    CONST robtarget T669:=[[77.479995,87.050626,11.799995],[0.000000,0.000000,1.000000,0.000000],[0,0,-1,0],[9E+09,9E+09,9E+09,9E+09,9E+09,9E+09]];
    CONST robtarget T670:=[[77.479995,72.949381,11.799995],[0.000000,0.000000,1.000000,0.000000],[0,0,-1,0],[9E+09,9E+09,9E+09,9E+09,9E+09,9E+09]];
    CONST robtarget T671:=[[77.479995,52.050624,11.799995],[0.000000,0.000000,1.000000,0.000000],[0,0,-1,0],[9E+09,9E+09,9E+09,9E+09,9E+09,9E+09]];
    CONST robtarget T672:=[[77.479995,37.949379,11.799995],[0.000000,0.000000,1.000000,0.000000],[0,0,-1,0],[9E+09,9E+09,9E+09,9E+09,9E+09,9E+09]];
    CONST robtarget T673:=[[77.479995,30.069007,11.799995],[0.000000,0.000000,1.000000,0.000000],[0,0,-1,0],[9E+09,9E+09,9E+09,9E+09,9E+09,9E+09]];
    CONST robtarget T674:=[[78.739999,30.028279,11.799995],[0.000000,0.000000,1.000000,0.000000],[0,0,-1,0],[9E+09,9E+09,9E+09,9E+09,9E+09,9E+09]];
    CONST robtarget T675:=[[78.739999,37.608991,11.799995],[0.000000,0.000000,1.000000,0.000000],[0,0,-1,0],[9E+09,9E+09,9E+09,9E+09,9E+09,9E+09]];
    CONST robtarget T676:=[[78.739999,52.391011,11.799995],[0.000000,0.000000,1.000000,0.000000],[0,0,-1,0],[9E+09,9E+09,9E+09,9E+09,9E+09,9E+09]];
    CONST robtarget T677:=[[78.739999,72.608994,11.799995],[0.000000,0.000000,1.000000,0.000000],[0,0,-1,0],[9E+09,9E+09,9E+09,9E+09,9E+09,9E+09]];
    CONST robtarget T678:=[[78.739999,87.391014,11.799995],[0.000000,0.000000,1.000000,0.000000],[0,0,-1,0],[9E+09,9E+09,9E+09,9E+09,9E+09,9E+09]];
    CONST robtarget T679:=[[78.739999,107.608996,11.799995],[0.000000,0.000000,1.000000,0.000000],[0,0,-1,0],[9E+09,9E+09,9E+09,9E+09,9E+09,9E+09]];
    CONST robtarget T680:=[[78.739999,122.391017,11.799995],[0.000000,0.000000,1.000000,0.000000],[0,0,-1,0],[9E+09,9E+09,9E+09,9E+09,9E+09,9E+09]];
    CONST robtarget T681:=[[78.739999,129.971729,11.799995],[0.000000,0.000000,1.000000,0.000000],[0,0,-1,0],[9E+09,9E+09,9E+09,9E+09,9E+09,9E+09]];
    CONST robtarget T682:=[[80.000004,130.000008,11.799995],[0.000000,0.000000,1.000000,0.000000],[0,0,-1,0],[9E+09,9E+09,9E+09,9E+09,9E+09,9E+09]];
    CONST robtarget T683:=[[80.000004,122.487319,11.799995],[0.000000,0.000000,1.000000,0.000000],[0,0,-1,0],[9E+09,9E+09,9E+09,9E+09,9E+09,9E+09]];
    CONST robtarget T684:=[[80.000004,107.512696,11.799995],[0.000000,0.000000,1.000000,0.000000],[0,0,-1,0],[9E+09,9E+09,9E+09,9E+09,9E+09,9E+09]];
    CONST robtarget T685:=[[80.000004,87.487316,11.799995],[0.000000,0.000000,1.000000,0.000000],[0,0,-1,0],[9E+09,9E+09,9E+09,9E+09,9E+09,9E+09]];
    CONST robtarget T686:=[[80.000004,72.512692,11.799995],[0.000000,0.000000,1.000000,0.000000],[0,0,-1,0],[9E+09,9E+09,9E+09,9E+09,9E+09,9E+09]];
    CONST robtarget T687:=[[80.000004,52.487312,11.799995],[0.000000,0.000000,1.000000,0.000000],[0,0,-1,0],[9E+09,9E+09,9E+09,9E+09,9E+09,9E+09]];
    CONST robtarget T688:=[[80.000004,37.512688,11.799995],[0.000000,0.000000,1.000000,0.000000],[0,0,-1,0],[9E+09,9E+09,9E+09,9E+09,9E+09,9E+09]];
    CONST robtarget T689:=[[80.000004,30.000000,11.799995],[0.000000,0.000000,1.000000,0.000000],[0,0,-1,0],[9E+09,9E+09,9E+09,9E+09,9E+09,9E+09]];
    CONST robtarget T690:=[[81.260008,30.028279,11.799995],[0.000000,0.000000,1.000000,0.000000],[0,0,-1,0],[9E+09,9E+09,9E+09,9E+09,9E+09,9E+09]];
    CONST robtarget T691:=[[81.260008,37.608991,11.799995],[0.000000,0.000000,1.000000,0.000000],[0,0,-1,0],[9E+09,9E+09,9E+09,9E+09,9E+09,9E+09]];
    CONST robtarget T692:=[[81.260008,52.391011,11.799995],[0.000000,0.000000,1.000000,0.000000],[0,0,-1,0],[9E+09,9E+09,9E+09,9E+09,9E+09,9E+09]];
    CONST robtarget T693:=[[81.260008,72.608994,11.799995],[0.000000,0.000000,1.000000,0.000000],[0,0,-1,0],[9E+09,9E+09,9E+09,9E+09,9E+09,9E+09]];
    CONST robtarget T694:=[[81.260008,87.391014,11.799995],[0.000000,0.000000,1.000000,0.000000],[0,0,-1,0],[9E+09,9E+09,9E+09,9E+09,9E+09,9E+09]];
    CONST robtarget T695:=[[81.260008,107.608996,11.799995],[0.000000,0.000000,1.000000,0.000000],[0,0,-1,0],[9E+09,9E+09,9E+09,9E+09,9E+09,9E+09]];
    CONST robtarget T696:=[[81.260008,122.391017,11.799995],[0.000000,0.000000,1.000000,0.000000],[0,0,-1,0],[9E+09,9E+09,9E+09,9E+09,9E+09,9E+09]];
    CONST robtarget T697:=[[81.260008,129.971729,11.799995],[0.000000,0.000000,1.000000,0.000000],[0,0,-1,0],[9E+09,9E+09,9E+09,9E+09,9E+09,9E+09]];
    CONST robtarget T698:=[[82.520013,129.931001,11.799995],[0.000000,0.000000,1.000000,0.000000],[0,0,-1,0],[9E+09,9E+09,9E+09,9E+09,9E+09,9E+09]];
    CONST robtarget T699:=[[82.520013,122.050628,11.799995],[0.000000,0.000000,1.000000,0.000000],[0,0,-1,0],[9E+09,9E+09,9E+09,9E+09,9E+09,9E+09]];
    CONST robtarget T700:=[[82.520013,107.949384,11.799995],[0.000000,0.000000,1.000000,0.000000],[0,0,-1,0],[9E+09,9E+09,9E+09,9E+09,9E+09,9E+09]];
    CONST robtarget T701:=[[82.520013,87.050626,11.799995],[0.000000,0.000000,1.000000,0.000000],[0,0,-1,0],[9E+09,9E+09,9E+09,9E+09,9E+09,9E+09]];
    CONST robtarget T702:=[[82.520013,72.949381,11.799995],[0.000000,0.000000,1.000000,0.000000],[0,0,-1,0],[9E+09,9E+09,9E+09,9E+09,9E+09,9E+09]];
    CONST robtarget T703:=[[82.520013,52.050624,11.799995],[0.000000,0.000000,1.000000,0.000000],[0,0,-1,0],[9E+09,9E+09,9E+09,9E+09,9E+09,9E+09]];
    CONST robtarget T704:=[[82.520013,37.949379,11.799995],[0.000000,0.000000,1.000000,0.000000],[0,0,-1,0],[9E+09,9E+09,9E+09,9E+09,9E+09,9E+09]];
    CONST robtarget T705:=[[82.520013,30.069007,11.799995],[0.000000,0.000000,1.000000,0.000000],[0,0,-1,0],[9E+09,9E+09,9E+09,9E+09,9E+09,9E+09]];
    CONST robtarget T706:=[[83.780017,30.153959,11.799995],[0.000000,0.000000,1.000000,0.000000],[0,0,-1,0],[9E+09,9E+09,9E+09,9E+09,9E+09,9E+09]];
    CONST robtarget T707:=[[83.780017,38.524551,11.799995],[0.000000,0.000000,1.000000,0.000000],[0,0,-1,0],[9E+09,9E+09,9E+09,9E+09,9E+09,9E+09]];
    CONST robtarget T708:=[[83.780017,51.475451,11.799995],[0.000000,0.000000,1.000000,0.000000],[0,0,-1,0],[9E+09,9E+09,9E+09,9E+09,9E+09,9E+09]];
    CONST robtarget T709:=[[83.780017,73.524553,11.799995],[0.000000,0.000000,1.000000,0.000000],[0,0,-1,0],[9E+09,9E+09,9E+09,9E+09,9E+09,9E+09]];
    CONST robtarget T710:=[[83.780017,86.475455,11.799995],[0.000000,0.000000,1.000000,0.000000],[0,0,-1,0],[9E+09,9E+09,9E+09,9E+09,9E+09,9E+09]];
    CONST robtarget T711:=[[83.780017,108.524556,11.799995],[0.000000,0.000000,1.000000,0.000000],[0,0,-1,0],[9E+09,9E+09,9E+09,9E+09,9E+09,9E+09]];
    CONST robtarget T712:=[[83.780017,121.475457,11.799995],[0.000000,0.000000,1.000000,0.000000],[0,0,-1,0],[9E+09,9E+09,9E+09,9E+09,9E+09,9E+09]];
    CONST robtarget T713:=[[83.780017,129.846049,11.799995],[0.000000,0.000000,1.000000,0.000000],[0,0,-1,0],[9E+09,9E+09,9E+09,9E+09,9E+09,9E+09]];
    CONST robtarget T714:=[[85.040022,129.735844,11.799995],[0.000000,0.000000,1.000000,0.000000],[0,0,-1,0],[9E+09,9E+09,9E+09,9E+09,9E+09,9E+09]];
    CONST robtarget T715:=[[85.040022,120.544921,11.799995],[0.000000,0.000000,1.000000,0.000000],[0,0,-1,0],[9E+09,9E+09,9E+09,9E+09,9E+09,9E+09]];
    CONST robtarget T716:=[[85.040022,109.455091,11.799995],[0.000000,0.000000,1.000000,0.000000],[0,0,-1,0],[9E+09,9E+09,9E+09,9E+09,9E+09,9E+09]];
    CONST robtarget T717:=[[85.040022,85.544918,11.799995],[0.000000,0.000000,1.000000,0.000000],[0,0,-1,0],[9E+09,9E+09,9E+09,9E+09,9E+09,9E+09]];
    CONST robtarget T718:=[[85.040022,74.455090,11.799995],[0.000000,0.000000,1.000000,0.000000],[0,0,-1,0],[9E+09,9E+09,9E+09,9E+09,9E+09,9E+09]];
    CONST robtarget T719:=[[85.040022,50.544916,11.799995],[0.000000,0.000000,1.000000,0.000000],[0,0,-1,0],[9E+09,9E+09,9E+09,9E+09,9E+09,9E+09]];
    CONST robtarget T720:=[[85.040022,39.455086,11.799995],[0.000000,0.000000,1.000000,0.000000],[0,0,-1,0],[9E+09,9E+09,9E+09,9E+09,9E+09,9E+09]];
    CONST robtarget T721:=[[85.040022,30.264163,11.799995],[0.000000,0.000000,1.000000,0.000000],[0,0,-1,0],[9E+09,9E+09,9E+09,9E+09,9E+09,9E+09]];
    CONST robtarget T722:=[[86.300026,30.406130,11.799995],[0.000000,0.000000,1.000000,0.000000],[0,0,-1,0],[9E+09,9E+09,9E+09,9E+09,9E+09,9E+09]];
    CONST robtarget T723:=[[86.300026,40.937335,11.799995],[0.000000,0.000000,1.000000,0.000000],[0,0,-1,0],[9E+09,9E+09,9E+09,9E+09,9E+09,9E+09]];
    CONST robtarget T724:=[[86.300026,49.062665,11.799995],[0.000000,0.000000,1.000000,0.000000],[0,0,-1,0],[9E+09,9E+09,9E+09,9E+09,9E+09,9E+09]];
    CONST robtarget T725:=[[86.300026,75.937339,11.799995],[0.000000,0.000000,1.000000,0.000000],[0,0,-1,0],[9E+09,9E+09,9E+09,9E+09,9E+09,9E+09]];
    CONST robtarget T726:=[[86.300026,84.062668,11.799995],[0.000000,0.000000,1.000000,0.000000],[0,0,-1,0],[9E+09,9E+09,9E+09,9E+09,9E+09,9E+09]];
    CONST robtarget T727:=[[86.300026,110.937342,11.799995],[0.000000,0.000000,1.000000,0.000000],[0,0,-1,0],[9E+09,9E+09,9E+09,9E+09,9E+09,9E+09]];
    CONST robtarget T728:=[[86.300026,119.062672,11.799995],[0.000000,0.000000,1.000000,0.000000],[0,0,-1,0],[9E+09,9E+09,9E+09,9E+09,9E+09,9E+09]];
    CONST robtarget T729:=[[86.300026,129.593877,11.799995],[0.000000,0.000000,1.000000,0.000000],[0,0,-1,0],[9E+09,9E+09,9E+09,9E+09,9E+09,9E+09]];
    CONST robtarget T730:=[[87.560031,129.413129,11.799995],[0.000000,0.000000,1.000000,0.000000],[0,0,-1,0],[9E+09,9E+09,9E+09,9E+09,9E+09,9E+09]];
    CONST robtarget T731:=[[87.560031,30.586879,11.799995],[0.000000,0.000000,1.000000,0.000000],[0,0,-1,0],[9E+09,9E+09,9E+09,9E+09,9E+09,9E+09]];
    CONST robtarget T732:=[[88.820035,30.786444,11.799995],[0.000000,0.000000,1.000000,0.000000],[0,0,-1,0],[9E+09,9E+09,9E+09,9E+09,9E+09,9E+09]];
    CONST robtarget T733:=[[88.820035,129.213563,11.799995],[0.000000,0.000000,1.000000,0.000000],[0,0,-1,0],[9E+09,9E+09,9E+09,9E+09,9E+09,9E+09]];
    CONST robtarget T734:=[[90.080040,128.960575,11.799995],[0.000000,0.000000,1.000000,0.000000],[0,0,-1,0],[9E+09,9E+09,9E+09,9E+09,9E+09,9E+09]];
    CONST robtarget T735:=[[90.080040,31.039433,11.799995],[0.000000,0.000000,1.000000,0.000000],[0,0,-1,0],[9E+09,9E+09,9E+09,9E+09,9E+09,9E+09]];
    CONST robtarget T736:=[[91.340044,31.307526,11.799995],[0.000000,0.000000,1.000000,0.000000],[0,0,-1,0],[9E+09,9E+09,9E+09,9E+09,9E+09,9E+09]];
    CONST robtarget T737:=[[91.340044,128.692481,11.799995],[0.000000,0.000000,1.000000,0.000000],[0,0,-1,0],[9E+09,9E+09,9E+09,9E+09,9E+09,9E+09]];
    CONST robtarget T738:=[[92.600049,128.374988,11.799995],[0.000000,0.000000,1.000000,0.000000],[0,0,-1,0],[9E+09,9E+09,9E+09,9E+09,9E+09,9E+09]];
    CONST robtarget T739:=[[92.600049,31.625019,11.799995],[0.000000,0.000000,1.000000,0.000000],[0,0,-1,0],[9E+09,9E+09,9E+09,9E+09,9E+09,9E+09]];
    CONST robtarget T740:=[[93.860053,31.969479,11.799995],[0.000000,0.000000,1.000000,0.000000],[0,0,-1,0],[9E+09,9E+09,9E+09,9E+09,9E+09,9E+09]];
    CONST robtarget T741:=[[93.860053,128.030529,11.799995],[0.000000,0.000000,1.000000,0.000000],[0,0,-1,0],[9E+09,9E+09,9E+09,9E+09,9E+09,9E+09]];
    CONST robtarget T742:=[[95.120058,127.652167,11.799995],[0.000000,0.000000,1.000000,0.000000],[0,0,-1,0],[9E+09,9E+09,9E+09,9E+09,9E+09,9E+09]];
    CONST robtarget T743:=[[95.120058,32.347841,11.799995],[0.000000,0.000000,1.000000,0.000000],[0,0,-1,0],[9E+09,9E+09,9E+09,9E+09,9E+09,9E+09]];
    CONST robtarget T744:=[[96.380062,32.772318,11.799995],[0.000000,0.000000,1.000000,0.000000],[0,0,-1,0],[9E+09,9E+09,9E+09,9E+09,9E+09,9E+09]];
    CONST robtarget T745:=[[96.380062,127.227690,11.799995],[0.000000,0.000000,1.000000,0.000000],[0,0,-1,0],[9E+09,9E+09,9E+09,9E+09,9E+09,9E+09]];
    CONST robtarget T746:=[[97.640067,126.783143,11.799995],[0.000000,0.000000,1.000000,0.000000],[0,0,-1,0],[9E+09,9E+09,9E+09,9E+09,9E+09,9E+09]];
    CONST robtarget T747:=[[97.640067,33.216864,11.799995],[0.000000,0.000000,1.000000,0.000000],[0,0,-1,0],[9E+09,9E+09,9E+09,9E+09,9E+09,9E+09]];
    CONST robtarget T748:=[[98.900071,33.722290,11.799995],[0.000000,0.000000,1.000000,0.000000],[0,0,-1,0],[9E+09,9E+09,9E+09,9E+09,9E+09,9E+09]];
    CONST robtarget T749:=[[98.900071,126.277717,11.799995],[0.000000,0.000000,1.000000,0.000000],[0,0,-1,0],[9E+09,9E+09,9E+09,9E+09,9E+09,9E+09]];
    CONST robtarget T750:=[[100.160076,125.745278,11.799995],[0.000000,0.000000,1.000000,0.000000],[0,0,-1,0],[9E+09,9E+09,9E+09,9E+09,9E+09,9E+09]];
    CONST robtarget T751:=[[100.160076,34.254730,11.799995],[0.000000,0.000000,1.000000,0.000000],[0,0,-1,0],[9E+09,9E+09,9E+09,9E+09,9E+09,9E+09]];
    CONST robtarget T752:=[[101.420080,34.827050,11.799995],[0.000000,0.000000,1.000000,0.000000],[0,0,-1,0],[9E+09,9E+09,9E+09,9E+09,9E+09,9E+09]];
    CONST robtarget T753:=[[101.420080,125.172958,11.799995],[0.000000,0.000000,1.000000,0.000000],[0,0,-1,0],[9E+09,9E+09,9E+09,9E+09,9E+09,9E+09]];
    CONST robtarget T754:=[[102.680085,124.546114,11.799995],[0.000000,0.000000,1.000000,0.000000],[0,0,-1,0],[9E+09,9E+09,9E+09,9E+09,9E+09,9E+09]];
    CONST robtarget T755:=[[102.680085,35.453894,11.799995],[0.000000,0.000000,1.000000,0.000000],[0,0,-1,0],[9E+09,9E+09,9E+09,9E+09,9E+09,9E+09]];
    CONST robtarget T756:=[[103.940089,36.110177,11.799995],[0.000000,0.000000,1.000000,0.000000],[0,0,-1,0],[9E+09,9E+09,9E+09,9E+09,9E+09,9E+09]];
    CONST robtarget T757:=[[103.940089,123.889831,11.799995],[0.000000,0.000000,1.000000,0.000000],[0,0,-1,0],[9E+09,9E+09,9E+09,9E+09,9E+09,9E+09]];
    CONST robtarget T758:=[[105.200094,123.174878,11.799995],[0.000000,0.000000,1.000000,0.000000],[0,0,-1,0],[9E+09,9E+09,9E+09,9E+09,9E+09,9E+09]];
    CONST robtarget T759:=[[105.200094,36.825129,11.799995],[0.000000,0.000000,1.000000,0.000000],[0,0,-1,0],[9E+09,9E+09,9E+09,9E+09,9E+09,9E+09]];
    CONST robtarget T760:=[[106.460098,37.589739,11.799995],[0.000000,0.000000,1.000000,0.000000],[0,0,-1,0],[9E+09,9E+09,9E+09,9E+09,9E+09,9E+09]];
    CONST robtarget T761:=[[106.460098,122.410268,11.799995],[0.000000,0.000000,1.000000,0.000000],[0,0,-1,0],[9E+09,9E+09,9E+09,9E+09,9E+09,9E+09]];
    CONST robtarget T762:=[[107.720103,121.607260,11.799995],[0.000000,0.000000,1.000000,0.000000],[0,0,-1,0],[9E+09,9E+09,9E+09,9E+09,9E+09,9E+09]];
    CONST robtarget T763:=[[107.720103,81.789524,11.799995],[0.000000,0.000000,1.000000,0.000000],[0,0,-1,0],[9E+09,9E+09,9E+09,9E+09,9E+09,9E+09]];
    CONST robtarget T764:=[[107.720103,78.210483,11.799995],[0.000000,0.000000,1.000000,0.000000],[0,0,-1,0],[9E+09,9E+09,9E+09,9E+09,9E+09,9E+09]];
    CONST robtarget T765:=[[107.720103,38.392748,11.799995],[0.000000,0.000000,1.000000,0.000000],[0,0,-1,0],[9E+09,9E+09,9E+09,9E+09,9E+09,9E+09]];
    CONST robtarget T766:=[[108.980107,39.265681,11.799995],[0.000000,0.000000,1.000000,0.000000],[0,0,-1,0],[9E+09,9E+09,9E+09,9E+09,9E+09,9E+09]];
    CONST robtarget T767:=[[108.980107,75.547902,11.799995],[0.000000,0.000000,1.000000,0.000000],[0,0,-1,0],[9E+09,9E+09,9E+09,9E+09,9E+09,9E+09]];
    CONST robtarget T768:=[[108.980107,84.452106,11.799995],[0.000000,0.000000,1.000000,0.000000],[0,0,-1,0],[9E+09,9E+09,9E+09,9E+09,9E+09,9E+09]];
    CONST robtarget T769:=[[108.980107,120.734326,11.799995],[0.000000,0.000000,1.000000,0.000000],[0,0,-1,0],[9E+09,9E+09,9E+09,9E+09,9E+09,9E+09]];
    CONST robtarget T770:=[[110.240112,119.803025,11.799995],[0.000000,0.000000,1.000000,0.000000],[0,0,-1,0],[9E+09,9E+09,9E+09,9E+09,9E+09,9E+09]];
    CONST robtarget T771:=[[110.240112,85.779969,11.799995],[0.000000,0.000000,1.000000,0.000000],[0,0,-1,0],[9E+09,9E+09,9E+09,9E+09,9E+09,9E+09]];
    CONST robtarget T772:=[[110.240112,74.220038,11.799995],[0.000000,0.000000,1.000000,0.000000],[0,0,-1,0],[9E+09,9E+09,9E+09,9E+09,9E+09,9E+09]];
    CONST robtarget T773:=[[110.240112,40.196983,11.799995],[0.000000,0.000000,1.000000,0.000000],[0,0,-1,0],[9E+09,9E+09,9E+09,9E+09,9E+09,9E+09]];
    CONST robtarget T774:=[[111.500116,41.180273,11.799995],[0.000000,0.000000,1.000000,0.000000],[0,0,-1,0],[9E+09,9E+09,9E+09,9E+09,9E+09,9E+09]];
    CONST robtarget T775:=[[111.500116,73.379202,11.799995],[0.000000,0.000000,1.000000,0.000000],[0,0,-1,0],[9E+09,9E+09,9E+09,9E+09,9E+09,9E+09]];
    CONST robtarget T776:=[[111.500116,86.620805,11.799995],[0.000000,0.000000,1.000000,0.000000],[0,0,-1,0],[9E+09,9E+09,9E+09,9E+09,9E+09,9E+09]];
    CONST robtarget T777:=[[111.500116,118.819735,11.799995],[0.000000,0.000000,1.000000,0.000000],[0,0,-1,0],[9E+09,9E+09,9E+09,9E+09,9E+09,9E+09]];
    CONST robtarget T778:=[[112.760121,117.767805,11.799995],[0.000000,0.000000,1.000000,0.000000],[0,0,-1,0],[9E+09,9E+09,9E+09,9E+09,9E+09,9E+09]];
    CONST robtarget T779:=[[112.760121,87.152583,11.799995],[0.000000,0.000000,1.000000,0.000000],[0,0,-1,0],[9E+09,9E+09,9E+09,9E+09,9E+09,9E+09]];
    CONST robtarget T780:=[[112.760121,72.847425,11.799995],[0.000000,0.000000,1.000000,0.000000],[0,0,-1,0],[9E+09,9E+09,9E+09,9E+09,9E+09,9E+09]];
    CONST robtarget T781:=[[112.760121,42.232203,11.799995],[0.000000,0.000000,1.000000,0.000000],[0,0,-1,0],[9E+09,9E+09,9E+09,9E+09,9E+09,9E+09]];
    CONST robtarget T782:=[[114.020125,43.373063,11.799995],[0.000000,0.000000,1.000000,0.000000],[0,0,-1,0],[9E+09,9E+09,9E+09,9E+09,9E+09,9E+09]];
    CONST robtarget T783:=[[114.020125,72.576253,11.799995],[0.000000,0.000000,1.000000,0.000000],[0,0,-1,0],[9E+09,9E+09,9E+09,9E+09,9E+09,9E+09]];
    CONST robtarget T784:=[[114.020125,87.423755,11.799995],[0.000000,0.000000,1.000000,0.000000],[0,0,-1,0],[9E+09,9E+09,9E+09,9E+09,9E+09,9E+09]];
    CONST robtarget T785:=[[114.020125,116.626944,11.799995],[0.000000,0.000000,1.000000,0.000000],[0,0,-1,0],[9E+09,9E+09,9E+09,9E+09,9E+09,9E+09]];
    CONST robtarget T786:=[[115.280130,115.412758,11.799995],[0.000000,0.000000,1.000000,0.000000],[0,0,-1,0],[9E+09,9E+09,9E+09,9E+09,9E+09,9E+09]];
    CONST robtarget T787:=[[115.280130,87.487316,11.799995],[0.000000,0.000000,1.000000,0.000000],[0,0,-1,0],[9E+09,9E+09,9E+09,9E+09,9E+09,9E+09]];
    CONST robtarget T788:=[[115.280130,72.512692,11.799995],[0.000000,0.000000,1.000000,0.000000],[0,0,-1,0],[9E+09,9E+09,9E+09,9E+09,9E+09,9E+09]];
    CONST robtarget T789:=[[115.280130,44.587250,11.799995],[0.000000,0.000000,1.000000,0.000000],[0,0,-1,0],[9E+09,9E+09,9E+09,9E+09,9E+09,9E+09]];
    CONST robtarget T790:=[[116.540134,45.884908,11.799995],[0.000000,0.000000,1.000000,0.000000],[0,0,-1,0],[9E+09,9E+09,9E+09,9E+09,9E+09,9E+09]];
    CONST robtarget T791:=[[116.540134,72.670297,11.799995],[0.000000,0.000000,1.000000,0.000000],[0,0,-1,0],[9E+09,9E+09,9E+09,9E+09,9E+09,9E+09]];
    CONST robtarget T792:=[[116.540134,87.329711,11.799995],[0.000000,0.000000,1.000000,0.000000],[0,0,-1,0],[9E+09,9E+09,9E+09,9E+09,9E+09,9E+09]];
    CONST robtarget T793:=[[116.540134,114.115099,11.799995],[0.000000,0.000000,1.000000,0.000000],[0,0,-1,0],[9E+09,9E+09,9E+09,9E+09,9E+09,9E+09]];
    CONST robtarget T794:=[[117.800139,112.721391,11.799995],[0.000000,0.000000,1.000000,0.000000],[0,0,-1,0],[9E+09,9E+09,9E+09,9E+09,9E+09,9E+09]];
    CONST robtarget T795:=[[117.800139,86.948670,11.799995],[0.000000,0.000000,1.000000,0.000000],[0,0,-1,0],[9E+09,9E+09,9E+09,9E+09,9E+09,9E+09]];
    CONST robtarget T796:=[[117.800139,73.051337,11.799995],[0.000000,0.000000,1.000000,0.000000],[0,0,-1,0],[9E+09,9E+09,9E+09,9E+09,9E+09,9E+09]];
    CONST robtarget T797:=[[117.800139,47.278617,11.799995],[0.000000,0.000000,1.000000,0.000000],[0,0,-1,0],[9E+09,9E+09,9E+09,9E+09,9E+09,9E+09]];
    CONST robtarget T798:=[[119.060143,48.787854,11.799995],[0.000000,0.000000,1.000000,0.000000],[0,0,-1,0],[9E+09,9E+09,9E+09,9E+09,9E+09,9E+09]];
    CONST robtarget T799:=[[119.060143,73.708792,11.799995],[0.000000,0.000000,1.000000,0.000000],[0,0,-1,0],[9E+09,9E+09,9E+09,9E+09,9E+09,9E+09]];
    CONST robtarget T800:=[[119.060143,86.291215,11.799995],[0.000000,0.000000,1.000000,0.000000],[0,0,-1,0],[9E+09,9E+09,9E+09,9E+09,9E+09,9E+09]];
    CONST robtarget T801:=[[119.060143,111.212154,11.799995],[0.000000,0.000000,1.000000,0.000000],[0,0,-1,0],[9E+09,9E+09,9E+09,9E+09,9E+09,9E+09]];
    CONST robtarget T802:=[[120.320148,109.560940,11.799995],[0.000000,0.000000,1.000000,0.000000],[0,0,-1,0],[9E+09,9E+09,9E+09,9E+09,9E+09,9E+09]];
    CONST robtarget T803:=[[120.320148,85.271589,11.799995],[0.000000,0.000000,1.000000,0.000000],[0,0,-1,0],[9E+09,9E+09,9E+09,9E+09,9E+09,9E+09]];
    CONST robtarget T804:=[[120.320148,74.728418,11.799995],[0.000000,0.000000,1.000000,0.000000],[0,0,-1,0],[9E+09,9E+09,9E+09,9E+09,9E+09,9E+09]];
    CONST robtarget T805:=[[120.320148,50.439068,11.799995],[0.000000,0.000000,1.000000,0.000000],[0,0,-1,0],[9E+09,9E+09,9E+09,9E+09,9E+09,9E+09]];
    CONST robtarget T806:=[[121.580152,52.240778,11.799995],[0.000000,0.000000,1.000000,0.000000],[0,0,-1,0],[9E+09,9E+09,9E+09,9E+09,9E+09,9E+09]];
    CONST robtarget T807:=[[121.580152,76.422528,11.799995],[0.000000,0.000000,1.000000,0.000000],[0,0,-1,0],[9E+09,9E+09,9E+09,9E+09,9E+09,9E+09]];
    CONST robtarget T808:=[[121.580152,83.577479,11.799995],[0.000000,0.000000,1.000000,0.000000],[0,0,-1,0],[9E+09,9E+09,9E+09,9E+09,9E+09,9E+09]];
    CONST robtarget T809:=[[121.580152,107.759230,11.799995],[0.000000,0.000000,1.000000,0.000000],[0,0,-1,0],[9E+09,9E+09,9E+09,9E+09,9E+09,9E+09]];
    CONST robtarget T810:=[[122.840157,105.775934,11.799995],[0.000000,0.000000,1.000000,0.000000],[0,0,-1,0],[9E+09,9E+09,9E+09,9E+09,9E+09,9E+09]];
    CONST robtarget T811:=[[122.840157,54.224074,11.799995],[0.000000,0.000000,1.000000,0.000000],[0,0,-1,0],[9E+09,9E+09,9E+09,9E+09,9E+09,9E+09]];
    CONST robtarget T812:=[[124.100161,56.444690,11.799995],[0.000000,0.000000,1.000000,0.000000],[0,0,-1,0],[9E+09,9E+09,9E+09,9E+09,9E+09,9E+09]];
    CONST robtarget T813:=[[124.100161,103.555317,11.799995],[0.000000,0.000000,1.000000,0.000000],[0,0,-1,0],[9E+09,9E+09,9E+09,9E+09,9E+09,9E+09]];
    CONST robtarget T814:=[[125.360166,101.007928,11.799995],[0.000000,0.000000,1.000000,0.000000],[0,0,-1,0],[9E+09,9E+09,9E+09,9E+09,9E+09,9E+09]];
    CONST robtarget T815:=[[125.360166,58.992080,11.799995],[0.000000,0.000000,1.000000,0.000000],[0,0,-1,0],[9E+09,9E+09,9E+09,9E+09,9E+09,9E+09]];
    CONST robtarget T816:=[[126.620170,61.953657,11.799995],[0.000000,0.000000,1.000000,0.000000],[0,0,-1,0],[9E+09,9E+09,9E+09,9E+09,9E+09,9E+09]];
    CONST robtarget T817:=[[126.620170,98.046351,11.799995],[0.000000,0.000000,1.000000,0.000000],[0,0,-1,0],[9E+09,9E+09,9E+09,9E+09,9E+09,9E+09]];
    CONST robtarget T818:=[[127.880175,94.360756,11.799995],[0.000000,0.000000,1.000000,0.000000],[0,0,-1,0],[9E+09,9E+09,9E+09,9E+09,9E+09,9E+09]];
    CONST robtarget T819:=[[127.880175,65.639251,11.799995],[0.000000,0.000000,1.000000,0.000000],[0,0,-1,0],[9E+09,9E+09,9E+09,9E+09,9E+09,9E+09]];
    CONST robtarget T820:=[[129.140179,70.797151,11.799995],[0.000000,0.000000,1.000000,0.000000],[0,0,-1,0],[9E+09,9E+09,9E+09,9E+09,9E+09,9E+09]];
    CONST robtarget T821:=[[129.140179,89.202857,11.799995],[0.000000,0.000000,1.000000,0.000000],[0,0,-1,0],[9E+09,9E+09,9E+09,9E+09,9E+09,9E+09]];
    CONST robtarget T822:=[[129.140179,70.797151,12.500005],[0.000000,0.000000,1.000000,0.000000],[0,0,-1,0],[9E+09,9E+09,9E+09,9E+09,9E+09,9E+09]];
    CONST robtarget T823:=[[129.140179,89.202857,12.500005],[0.000000,0.000000,1.000000,0.000000],[0,0,-1,0],[9E+09,9E+09,9E+09,9E+09,9E+09,9E+09]];
    CONST robtarget T824:=[[129.140179,70.797151,12.500005],[0.000000,0.000000,1.000000,0.000000],[0,0,-1,0],[9E+09,9E+09,9E+09,9E+09,9E+09,9E+09]];
    CONST robtarget T825:=[[129.140179,89.202857,12.500005],[0.000000,0.000000,1.000000,0.000000],[0,0,-1,0],[9E+09,9E+09,9E+09,9E+09,9E+09,9E+09]];
    CONST robtarget T826:=[[127.880175,94.360756,12.500005],[0.000000,0.000000,1.000000,0.000000],[0,0,-1,0],[9E+09,9E+09,9E+09,9E+09,9E+09,9E+09]];
    CONST robtarget T827:=[[127.880175,65.639251,12.500005],[0.000000,0.000000,1.000000,0.000000],[0,0,-1,0],[9E+09,9E+09,9E+09,9E+09,9E+09,9E+09]];
    CONST robtarget T828:=[[126.620170,61.953657,12.500005],[0.000000,0.000000,1.000000,0.000000],[0,0,-1,0],[9E+09,9E+09,9E+09,9E+09,9E+09,9E+09]];
    CONST robtarget T829:=[[126.620170,98.046351,12.500005],[0.000000,0.000000,1.000000,0.000000],[0,0,-1,0],[9E+09,9E+09,9E+09,9E+09,9E+09,9E+09]];
    CONST robtarget T830:=[[125.360166,101.007928,12.500005],[0.000000,0.000000,1.000000,0.000000],[0,0,-1,0],[9E+09,9E+09,9E+09,9E+09,9E+09,9E+09]];
    CONST robtarget T831:=[[125.360166,58.992080,12.500005],[0.000000,0.000000,1.000000,0.000000],[0,0,-1,0],[9E+09,9E+09,9E+09,9E+09,9E+09,9E+09]];
    CONST robtarget T832:=[[124.100161,56.444690,12.500005],[0.000000,0.000000,1.000000,0.000000],[0,0,-1,0],[9E+09,9E+09,9E+09,9E+09,9E+09,9E+09]];
    CONST robtarget T833:=[[124.100161,103.555317,12.500005],[0.000000,0.000000,1.000000,0.000000],[0,0,-1,0],[9E+09,9E+09,9E+09,9E+09,9E+09,9E+09]];
    CONST robtarget T834:=[[122.840157,105.775934,12.500005],[0.000000,0.000000,1.000000,0.000000],[0,0,-1,0],[9E+09,9E+09,9E+09,9E+09,9E+09,9E+09]];
    CONST robtarget T835:=[[122.840157,54.224074,12.500005],[0.000000,0.000000,1.000000,0.000000],[0,0,-1,0],[9E+09,9E+09,9E+09,9E+09,9E+09,9E+09]];
    CONST robtarget T836:=[[121.580152,52.240778,12.500005],[0.000000,0.000000,1.000000,0.000000],[0,0,-1,0],[9E+09,9E+09,9E+09,9E+09,9E+09,9E+09]];
    CONST robtarget T837:=[[121.580152,76.422528,12.500005],[0.000000,0.000000,1.000000,0.000000],[0,0,-1,0],[9E+09,9E+09,9E+09,9E+09,9E+09,9E+09]];
    CONST robtarget T838:=[[121.580152,83.577479,12.500005],[0.000000,0.000000,1.000000,0.000000],[0,0,-1,0],[9E+09,9E+09,9E+09,9E+09,9E+09,9E+09]];
    CONST robtarget T839:=[[121.580152,107.759230,12.500005],[0.000000,0.000000,1.000000,0.000000],[0,0,-1,0],[9E+09,9E+09,9E+09,9E+09,9E+09,9E+09]];
    CONST robtarget T840:=[[120.320148,109.560940,12.500005],[0.000000,0.000000,1.000000,0.000000],[0,0,-1,0],[9E+09,9E+09,9E+09,9E+09,9E+09,9E+09]];
    CONST robtarget T841:=[[120.320148,85.271589,12.500005],[0.000000,0.000000,1.000000,0.000000],[0,0,-1,0],[9E+09,9E+09,9E+09,9E+09,9E+09,9E+09]];
    CONST robtarget T842:=[[120.320148,74.728418,12.500005],[0.000000,0.000000,1.000000,0.000000],[0,0,-1,0],[9E+09,9E+09,9E+09,9E+09,9E+09,9E+09]];
    CONST robtarget T843:=[[120.320148,50.439068,12.500005],[0.000000,0.000000,1.000000,0.000000],[0,0,-1,0],[9E+09,9E+09,9E+09,9E+09,9E+09,9E+09]];
    CONST robtarget T844:=[[119.060143,48.787854,12.500005],[0.000000,0.000000,1.000000,0.000000],[0,0,-1,0],[9E+09,9E+09,9E+09,9E+09,9E+09,9E+09]];
    CONST robtarget T845:=[[119.060143,73.708792,12.500005],[0.000000,0.000000,1.000000,0.000000],[0,0,-1,0],[9E+09,9E+09,9E+09,9E+09,9E+09,9E+09]];
    CONST robtarget T846:=[[119.060143,86.291215,12.500005],[0.000000,0.000000,1.000000,0.000000],[0,0,-1,0],[9E+09,9E+09,9E+09,9E+09,9E+09,9E+09]];
    CONST robtarget T847:=[[119.060143,111.212154,12.500005],[0.000000,0.000000,1.000000,0.000000],[0,0,-1,0],[9E+09,9E+09,9E+09,9E+09,9E+09,9E+09]];
    CONST robtarget T848:=[[117.800139,112.721391,12.500005],[0.000000,0.000000,1.000000,0.000000],[0,0,-1,0],[9E+09,9E+09,9E+09,9E+09,9E+09,9E+09]];
    CONST robtarget T849:=[[117.800139,86.948670,12.500005],[0.000000,0.000000,1.000000,0.000000],[0,0,-1,0],[9E+09,9E+09,9E+09,9E+09,9E+09,9E+09]];
    CONST robtarget T850:=[[117.800139,73.051337,12.500005],[0.000000,0.000000,1.000000,0.000000],[0,0,-1,0],[9E+09,9E+09,9E+09,9E+09,9E+09,9E+09]];
    CONST robtarget T851:=[[117.800139,47.278617,12.500005],[0.000000,0.000000,1.000000,0.000000],[0,0,-1,0],[9E+09,9E+09,9E+09,9E+09,9E+09,9E+09]];
    CONST robtarget T852:=[[116.540134,45.884908,12.500005],[0.000000,0.000000,1.000000,0.000000],[0,0,-1,0],[9E+09,9E+09,9E+09,9E+09,9E+09,9E+09]];
    CONST robtarget T853:=[[116.540134,72.670297,12.500005],[0.000000,0.000000,1.000000,0.000000],[0,0,-1,0],[9E+09,9E+09,9E+09,9E+09,9E+09,9E+09]];
    CONST robtarget T854:=[[116.540134,87.329711,12.500005],[0.000000,0.000000,1.000000,0.000000],[0,0,-1,0],[9E+09,9E+09,9E+09,9E+09,9E+09,9E+09]];
    CONST robtarget T855:=[[116.540134,114.115099,12.500005],[0.000000,0.000000,1.000000,0.000000],[0,0,-1,0],[9E+09,9E+09,9E+09,9E+09,9E+09,9E+09]];
    CONST robtarget T856:=[[115.280130,115.412758,12.500005],[0.000000,0.000000,1.000000,0.000000],[0,0,-1,0],[9E+09,9E+09,9E+09,9E+09,9E+09,9E+09]];
    CONST robtarget T857:=[[115.280130,87.487316,12.500005],[0.000000,0.000000,1.000000,0.000000],[0,0,-1,0],[9E+09,9E+09,9E+09,9E+09,9E+09,9E+09]];
    CONST robtarget T858:=[[115.280130,72.512692,12.500005],[0.000000,0.000000,1.000000,0.000000],[0,0,-1,0],[9E+09,9E+09,9E+09,9E+09,9E+09,9E+09]];
    CONST robtarget T859:=[[115.280130,44.587250,12.500005],[0.000000,0.000000,1.000000,0.000000],[0,0,-1,0],[9E+09,9E+09,9E+09,9E+09,9E+09,9E+09]];
    CONST robtarget T860:=[[114.020125,43.373063,12.500005],[0.000000,0.000000,1.000000,0.000000],[0,0,-1,0],[9E+09,9E+09,9E+09,9E+09,9E+09,9E+09]];
    CONST robtarget T861:=[[114.020125,72.576253,12.500005],[0.000000,0.000000,1.000000,0.000000],[0,0,-1,0],[9E+09,9E+09,9E+09,9E+09,9E+09,9E+09]];
    CONST robtarget T862:=[[114.020125,87.423755,12.500005],[0.000000,0.000000,1.000000,0.000000],[0,0,-1,0],[9E+09,9E+09,9E+09,9E+09,9E+09,9E+09]];
    CONST robtarget T863:=[[114.020125,116.626944,12.500005],[0.000000,0.000000,1.000000,0.000000],[0,0,-1,0],[9E+09,9E+09,9E+09,9E+09,9E+09,9E+09]];
    CONST robtarget T864:=[[112.760121,117.767805,12.500005],[0.000000,0.000000,1.000000,0.000000],[0,0,-1,0],[9E+09,9E+09,9E+09,9E+09,9E+09,9E+09]];
    CONST robtarget T865:=[[112.760121,87.152583,12.500005],[0.000000,0.000000,1.000000,0.000000],[0,0,-1,0],[9E+09,9E+09,9E+09,9E+09,9E+09,9E+09]];
    CONST robtarget T866:=[[112.760121,72.847425,12.500005],[0.000000,0.000000,1.000000,0.000000],[0,0,-1,0],[9E+09,9E+09,9E+09,9E+09,9E+09,9E+09]];
    CONST robtarget T867:=[[112.760121,42.232203,12.500005],[0.000000,0.000000,1.000000,0.000000],[0,0,-1,0],[9E+09,9E+09,9E+09,9E+09,9E+09,9E+09]];
    CONST robtarget T868:=[[111.500116,41.180273,12.500005],[0.000000,0.000000,1.000000,0.000000],[0,0,-1,0],[9E+09,9E+09,9E+09,9E+09,9E+09,9E+09]];
    CONST robtarget T869:=[[111.500116,73.379202,12.500005],[0.000000,0.000000,1.000000,0.000000],[0,0,-1,0],[9E+09,9E+09,9E+09,9E+09,9E+09,9E+09]];
    CONST robtarget T870:=[[111.500116,86.620805,12.500005],[0.000000,0.000000,1.000000,0.000000],[0,0,-1,0],[9E+09,9E+09,9E+09,9E+09,9E+09,9E+09]];
    CONST robtarget T871:=[[111.500116,118.819735,12.500005],[0.000000,0.000000,1.000000,0.000000],[0,0,-1,0],[9E+09,9E+09,9E+09,9E+09,9E+09,9E+09]];
    CONST robtarget T872:=[[110.240112,119.803025,12.500005],[0.000000,0.000000,1.000000,0.000000],[0,0,-1,0],[9E+09,9E+09,9E+09,9E+09,9E+09,9E+09]];
    CONST robtarget T873:=[[110.240112,85.779969,12.500005],[0.000000,0.000000,1.000000,0.000000],[0,0,-1,0],[9E+09,9E+09,9E+09,9E+09,9E+09,9E+09]];
    CONST robtarget T874:=[[110.240112,74.220038,12.500005],[0.000000,0.000000,1.000000,0.000000],[0,0,-1,0],[9E+09,9E+09,9E+09,9E+09,9E+09,9E+09]];
    CONST robtarget T875:=[[110.240112,40.196983,12.500005],[0.000000,0.000000,1.000000,0.000000],[0,0,-1,0],[9E+09,9E+09,9E+09,9E+09,9E+09,9E+09]];
    CONST robtarget T876:=[[108.980107,39.265681,12.500005],[0.000000,0.000000,1.000000,0.000000],[0,0,-1,0],[9E+09,9E+09,9E+09,9E+09,9E+09,9E+09]];
    CONST robtarget T877:=[[108.980107,75.547902,12.500005],[0.000000,0.000000,1.000000,0.000000],[0,0,-1,0],[9E+09,9E+09,9E+09,9E+09,9E+09,9E+09]];
    CONST robtarget T878:=[[108.980107,84.452106,12.500005],[0.000000,0.000000,1.000000,0.000000],[0,0,-1,0],[9E+09,9E+09,9E+09,9E+09,9E+09,9E+09]];
    CONST robtarget T879:=[[108.980107,120.734326,12.500005],[0.000000,0.000000,1.000000,0.000000],[0,0,-1,0],[9E+09,9E+09,9E+09,9E+09,9E+09,9E+09]];
    CONST robtarget T880:=[[107.720103,121.607260,12.500005],[0.000000,0.000000,1.000000,0.000000],[0,0,-1,0],[9E+09,9E+09,9E+09,9E+09,9E+09,9E+09]];
    CONST robtarget T881:=[[107.720103,81.789524,12.500005],[0.000000,0.000000,1.000000,0.000000],[0,0,-1,0],[9E+09,9E+09,9E+09,9E+09,9E+09,9E+09]];
    CONST robtarget T882:=[[107.720103,78.210483,12.500005],[0.000000,0.000000,1.000000,0.000000],[0,0,-1,0],[9E+09,9E+09,9E+09,9E+09,9E+09,9E+09]];
    CONST robtarget T883:=[[107.720103,38.392748,12.500005],[0.000000,0.000000,1.000000,0.000000],[0,0,-1,0],[9E+09,9E+09,9E+09,9E+09,9E+09,9E+09]];
    CONST robtarget T884:=[[106.460098,37.589739,12.500005],[0.000000,0.000000,1.000000,0.000000],[0,0,-1,0],[9E+09,9E+09,9E+09,9E+09,9E+09,9E+09]];
    CONST robtarget T885:=[[106.460098,122.410268,12.500005],[0.000000,0.000000,1.000000,0.000000],[0,0,-1,0],[9E+09,9E+09,9E+09,9E+09,9E+09,9E+09]];
    CONST robtarget T886:=[[105.200094,123.174878,12.500005],[0.000000,0.000000,1.000000,0.000000],[0,0,-1,0],[9E+09,9E+09,9E+09,9E+09,9E+09,9E+09]];
    CONST robtarget T887:=[[105.200094,36.825129,12.500005],[0.000000,0.000000,1.000000,0.000000],[0,0,-1,0],[9E+09,9E+09,9E+09,9E+09,9E+09,9E+09]];
    CONST robtarget T888:=[[103.940089,36.110177,12.500005],[0.000000,0.000000,1.000000,0.000000],[0,0,-1,0],[9E+09,9E+09,9E+09,9E+09,9E+09,9E+09]];
    CONST robtarget T889:=[[103.940089,123.889831,12.500005],[0.000000,0.000000,1.000000,0.000000],[0,0,-1,0],[9E+09,9E+09,9E+09,9E+09,9E+09,9E+09]];
    CONST robtarget T890:=[[102.680085,124.546114,12.500005],[0.000000,0.000000,1.000000,0.000000],[0,0,-1,0],[9E+09,9E+09,9E+09,9E+09,9E+09,9E+09]];
    CONST robtarget T891:=[[102.680085,35.453894,12.500005],[0.000000,0.000000,1.000000,0.000000],[0,0,-1,0],[9E+09,9E+09,9E+09,9E+09,9E+09,9E+09]];
    CONST robtarget T892:=[[101.420080,34.827050,12.500005],[0.000000,0.000000,1.000000,0.000000],[0,0,-1,0],[9E+09,9E+09,9E+09,9E+09,9E+09,9E+09]];
    CONST robtarget T893:=[[101.420080,125.172958,12.500005],[0.000000,0.000000,1.000000,0.000000],[0,0,-1,0],[9E+09,9E+09,9E+09,9E+09,9E+09,9E+09]];
    CONST robtarget T894:=[[100.160076,125.745278,12.500005],[0.000000,0.000000,1.000000,0.000000],[0,0,-1,0],[9E+09,9E+09,9E+09,9E+09,9E+09,9E+09]];
    CONST robtarget T895:=[[100.160076,34.254730,12.500005],[0.000000,0.000000,1.000000,0.000000],[0,0,-1,0],[9E+09,9E+09,9E+09,9E+09,9E+09,9E+09]];
    CONST robtarget T896:=[[98.900071,33.722290,12.500005],[0.000000,0.000000,1.000000,0.000000],[0,0,-1,0],[9E+09,9E+09,9E+09,9E+09,9E+09,9E+09]];
    CONST robtarget T897:=[[98.900071,126.277717,12.500005],[0.000000,0.000000,1.000000,0.000000],[0,0,-1,0],[9E+09,9E+09,9E+09,9E+09,9E+09,9E+09]];
    CONST robtarget T898:=[[97.640067,126.783143,12.500005],[0.000000,0.000000,1.000000,0.000000],[0,0,-1,0],[9E+09,9E+09,9E+09,9E+09,9E+09,9E+09]];
    CONST robtarget T899:=[[97.640067,33.216864,12.500005],[0.000000,0.000000,1.000000,0.000000],[0,0,-1,0],[9E+09,9E+09,9E+09,9E+09,9E+09,9E+09]];
    CONST robtarget T900:=[[96.380062,32.772318,12.500005],[0.000000,0.000000,1.000000,0.000000],[0,0,-1,0],[9E+09,9E+09,9E+09,9E+09,9E+09,9E+09]];
    CONST robtarget T901:=[[96.380062,127.227690,12.500005],[0.000000,0.000000,1.000000,0.000000],[0,0,-1,0],[9E+09,9E+09,9E+09,9E+09,9E+09,9E+09]];
    CONST robtarget T902:=[[95.120058,127.652167,12.500005],[0.000000,0.000000,1.000000,0.000000],[0,0,-1,0],[9E+09,9E+09,9E+09,9E+09,9E+09,9E+09]];
    CONST robtarget T903:=[[95.120058,32.347841,12.500005],[0.000000,0.000000,1.000000,0.000000],[0,0,-1,0],[9E+09,9E+09,9E+09,9E+09,9E+09,9E+09]];
    CONST robtarget T904:=[[93.860053,31.969479,12.500005],[0.000000,0.000000,1.000000,0.000000],[0,0,-1,0],[9E+09,9E+09,9E+09,9E+09,9E+09,9E+09]];
    CONST robtarget T905:=[[93.860053,128.030529,12.500005],[0.000000,0.000000,1.000000,0.000000],[0,0,-1,0],[9E+09,9E+09,9E+09,9E+09,9E+09,9E+09]];
    CONST robtarget T906:=[[92.600049,128.374988,12.500005],[0.000000,0.000000,1.000000,0.000000],[0,0,-1,0],[9E+09,9E+09,9E+09,9E+09,9E+09,9E+09]];
    CONST robtarget T907:=[[92.600049,31.625019,12.500005],[0.000000,0.000000,1.000000,0.000000],[0,0,-1,0],[9E+09,9E+09,9E+09,9E+09,9E+09,9E+09]];
    CONST robtarget T908:=[[91.340044,31.307526,12.500005],[0.000000,0.000000,1.000000,0.000000],[0,0,-1,0],[9E+09,9E+09,9E+09,9E+09,9E+09,9E+09]];
    CONST robtarget T909:=[[91.340044,128.692481,12.500005],[0.000000,0.000000,1.000000,0.000000],[0,0,-1,0],[9E+09,9E+09,9E+09,9E+09,9E+09,9E+09]];
    CONST robtarget T910:=[[90.080040,128.960575,12.500005],[0.000000,0.000000,1.000000,0.000000],[0,0,-1,0],[9E+09,9E+09,9E+09,9E+09,9E+09,9E+09]];
    CONST robtarget T911:=[[90.080040,31.039433,12.500005],[0.000000,0.000000,1.000000,0.000000],[0,0,-1,0],[9E+09,9E+09,9E+09,9E+09,9E+09,9E+09]];
    CONST robtarget T912:=[[88.820035,30.786444,12.500005],[0.000000,0.000000,1.000000,0.000000],[0,0,-1,0],[9E+09,9E+09,9E+09,9E+09,9E+09,9E+09]];
    CONST robtarget T913:=[[88.820035,129.213563,12.500005],[0.000000,0.000000,1.000000,0.000000],[0,0,-1,0],[9E+09,9E+09,9E+09,9E+09,9E+09,9E+09]];
    CONST robtarget T914:=[[87.560031,129.413129,12.500005],[0.000000,0.000000,1.000000,0.000000],[0,0,-1,0],[9E+09,9E+09,9E+09,9E+09,9E+09,9E+09]];
    CONST robtarget T915:=[[87.560031,30.586879,12.500005],[0.000000,0.000000,1.000000,0.000000],[0,0,-1,0],[9E+09,9E+09,9E+09,9E+09,9E+09,9E+09]];
    CONST robtarget T916:=[[86.300026,30.406130,12.500005],[0.000000,0.000000,1.000000,0.000000],[0,0,-1,0],[9E+09,9E+09,9E+09,9E+09,9E+09,9E+09]];
    CONST robtarget T917:=[[86.300026,40.937335,12.500005],[0.000000,0.000000,1.000000,0.000000],[0,0,-1,0],[9E+09,9E+09,9E+09,9E+09,9E+09,9E+09]];
    CONST robtarget T918:=[[86.300026,49.062665,12.500005],[0.000000,0.000000,1.000000,0.000000],[0,0,-1,0],[9E+09,9E+09,9E+09,9E+09,9E+09,9E+09]];
    CONST robtarget T919:=[[86.300026,75.937339,12.500005],[0.000000,0.000000,1.000000,0.000000],[0,0,-1,0],[9E+09,9E+09,9E+09,9E+09,9E+09,9E+09]];
    CONST robtarget T920:=[[86.300026,84.062668,12.500005],[0.000000,0.000000,1.000000,0.000000],[0,0,-1,0],[9E+09,9E+09,9E+09,9E+09,9E+09,9E+09]];
    CONST robtarget T921:=[[86.300026,110.937342,12.500005],[0.000000,0.000000,1.000000,0.000000],[0,0,-1,0],[9E+09,9E+09,9E+09,9E+09,9E+09,9E+09]];
    CONST robtarget T922:=[[86.300026,119.062672,12.500005],[0.000000,0.000000,1.000000,0.000000],[0,0,-1,0],[9E+09,9E+09,9E+09,9E+09,9E+09,9E+09]];
    CONST robtarget T923:=[[86.300026,129.593877,12.500005],[0.000000,0.000000,1.000000,0.000000],[0,0,-1,0],[9E+09,9E+09,9E+09,9E+09,9E+09,9E+09]];
    CONST robtarget T924:=[[85.040022,129.735844,12.500005],[0.000000,0.000000,1.000000,0.000000],[0,0,-1,0],[9E+09,9E+09,9E+09,9E+09,9E+09,9E+09]];
    CONST robtarget T925:=[[85.040022,120.544921,12.500005],[0.000000,0.000000,1.000000,0.000000],[0,0,-1,0],[9E+09,9E+09,9E+09,9E+09,9E+09,9E+09]];
    CONST robtarget T926:=[[85.040022,109.455091,12.500005],[0.000000,0.000000,1.000000,0.000000],[0,0,-1,0],[9E+09,9E+09,9E+09,9E+09,9E+09,9E+09]];
    CONST robtarget T927:=[[85.040022,85.544918,12.500005],[0.000000,0.000000,1.000000,0.000000],[0,0,-1,0],[9E+09,9E+09,9E+09,9E+09,9E+09,9E+09]];
    CONST robtarget T928:=[[85.040022,74.455090,12.500005],[0.000000,0.000000,1.000000,0.000000],[0,0,-1,0],[9E+09,9E+09,9E+09,9E+09,9E+09,9E+09]];
    CONST robtarget T929:=[[85.040022,50.544916,12.500005],[0.000000,0.000000,1.000000,0.000000],[0,0,-1,0],[9E+09,9E+09,9E+09,9E+09,9E+09,9E+09]];
    CONST robtarget T930:=[[85.040022,39.455086,12.500005],[0.000000,0.000000,1.000000,0.000000],[0,0,-1,0],[9E+09,9E+09,9E+09,9E+09,9E+09,9E+09]];
    CONST robtarget T931:=[[85.040022,30.264163,12.500005],[0.000000,0.000000,1.000000,0.000000],[0,0,-1,0],[9E+09,9E+09,9E+09,9E+09,9E+09,9E+09]];
    CONST robtarget T932:=[[83.780017,30.153959,12.500005],[0.000000,0.000000,1.000000,0.000000],[0,0,-1,0],[9E+09,9E+09,9E+09,9E+09,9E+09,9E+09]];
    CONST robtarget T933:=[[83.780017,38.524551,12.500005],[0.000000,0.000000,1.000000,0.000000],[0,0,-1,0],[9E+09,9E+09,9E+09,9E+09,9E+09,9E+09]];
    CONST robtarget T934:=[[83.780017,51.475451,12.500005],[0.000000,0.000000,1.000000,0.000000],[0,0,-1,0],[9E+09,9E+09,9E+09,9E+09,9E+09,9E+09]];
    CONST robtarget T935:=[[83.780017,73.524553,12.500005],[0.000000,0.000000,1.000000,0.000000],[0,0,-1,0],[9E+09,9E+09,9E+09,9E+09,9E+09,9E+09]];
    CONST robtarget T936:=[[83.780017,86.475455,12.500005],[0.000000,0.000000,1.000000,0.000000],[0,0,-1,0],[9E+09,9E+09,9E+09,9E+09,9E+09,9E+09]];
    CONST robtarget T937:=[[83.780017,108.524556,12.500005],[0.000000,0.000000,1.000000,0.000000],[0,0,-1,0],[9E+09,9E+09,9E+09,9E+09,9E+09,9E+09]];
    CONST robtarget T938:=[[83.780017,121.475457,12.500005],[0.000000,0.000000,1.000000,0.000000],[0,0,-1,0],[9E+09,9E+09,9E+09,9E+09,9E+09,9E+09]];
    CONST robtarget T939:=[[83.780017,129.846049,12.500005],[0.000000,0.000000,1.000000,0.000000],[0,0,-1,0],[9E+09,9E+09,9E+09,9E+09,9E+09,9E+09]];
    CONST robtarget T940:=[[82.520013,129.931001,12.500005],[0.000000,0.000000,1.000000,0.000000],[0,0,-1,0],[9E+09,9E+09,9E+09,9E+09,9E+09,9E+09]];
    CONST robtarget T941:=[[82.520013,122.050628,12.500005],[0.000000,0.000000,1.000000,0.000000],[0,0,-1,0],[9E+09,9E+09,9E+09,9E+09,9E+09,9E+09]];
    CONST robtarget T942:=[[82.520013,107.949384,12.500005],[0.000000,0.000000,1.000000,0.000000],[0,0,-1,0],[9E+09,9E+09,9E+09,9E+09,9E+09,9E+09]];
    CONST robtarget T943:=[[82.520013,87.050626,12.500005],[0.000000,0.000000,1.000000,0.000000],[0,0,-1,0],[9E+09,9E+09,9E+09,9E+09,9E+09,9E+09]];
    CONST robtarget T944:=[[82.520013,72.949381,12.500005],[0.000000,0.000000,1.000000,0.000000],[0,0,-1,0],[9E+09,9E+09,9E+09,9E+09,9E+09,9E+09]];
    CONST robtarget T945:=[[82.520013,52.050624,12.500005],[0.000000,0.000000,1.000000,0.000000],[0,0,-1,0],[9E+09,9E+09,9E+09,9E+09,9E+09,9E+09]];
    CONST robtarget T946:=[[82.520013,37.949379,12.500005],[0.000000,0.000000,1.000000,0.000000],[0,0,-1,0],[9E+09,9E+09,9E+09,9E+09,9E+09,9E+09]];
    CONST robtarget T947:=[[82.520013,30.069007,12.500005],[0.000000,0.000000,1.000000,0.000000],[0,0,-1,0],[9E+09,9E+09,9E+09,9E+09,9E+09,9E+09]];
    CONST robtarget T948:=[[81.260008,30.028279,12.500005],[0.000000,0.000000,1.000000,0.000000],[0,0,-1,0],[9E+09,9E+09,9E+09,9E+09,9E+09,9E+09]];
    CONST robtarget T949:=[[81.260008,37.608991,12.500005],[0.000000,0.000000,1.000000,0.000000],[0,0,-1,0],[9E+09,9E+09,9E+09,9E+09,9E+09,9E+09]];
    CONST robtarget T950:=[[81.260008,52.391011,12.500005],[0.000000,0.000000,1.000000,0.000000],[0,0,-1,0],[9E+09,9E+09,9E+09,9E+09,9E+09,9E+09]];
    CONST robtarget T951:=[[81.260008,72.608994,12.500005],[0.000000,0.000000,1.000000,0.000000],[0,0,-1,0],[9E+09,9E+09,9E+09,9E+09,9E+09,9E+09]];
    CONST robtarget T952:=[[81.260008,87.391014,12.500005],[0.000000,0.000000,1.000000,0.000000],[0,0,-1,0],[9E+09,9E+09,9E+09,9E+09,9E+09,9E+09]];
    CONST robtarget T953:=[[81.260008,107.608996,12.500005],[0.000000,0.000000,1.000000,0.000000],[0,0,-1,0],[9E+09,9E+09,9E+09,9E+09,9E+09,9E+09]];
    CONST robtarget T954:=[[81.260008,122.391017,12.500005],[0.000000,0.000000,1.000000,0.000000],[0,0,-1,0],[9E+09,9E+09,9E+09,9E+09,9E+09,9E+09]];
    CONST robtarget T955:=[[81.260008,129.971729,12.500005],[0.000000,0.000000,1.000000,0.000000],[0,0,-1,0],[9E+09,9E+09,9E+09,9E+09,9E+09,9E+09]];
    CONST robtarget T956:=[[80.000004,130.000008,12.500005],[0.000000,0.000000,1.000000,0.000000],[0,0,-1,0],[9E+09,9E+09,9E+09,9E+09,9E+09,9E+09]];
    CONST robtarget T957:=[[80.000004,122.487319,12.500005],[0.000000,0.000000,1.000000,0.000000],[0,0,-1,0],[9E+09,9E+09,9E+09,9E+09,9E+09,9E+09]];
    CONST robtarget T958:=[[80.000004,107.512696,12.500005],[0.000000,0.000000,1.000000,0.000000],[0,0,-1,0],[9E+09,9E+09,9E+09,9E+09,9E+09,9E+09]];
    CONST robtarget T959:=[[80.000004,87.487316,12.500005],[0.000000,0.000000,1.000000,0.000000],[0,0,-1,0],[9E+09,9E+09,9E+09,9E+09,9E+09,9E+09]];
    CONST robtarget T960:=[[80.000004,72.512692,12.500005],[0.000000,0.000000,1.000000,0.000000],[0,0,-1,0],[9E+09,9E+09,9E+09,9E+09,9E+09,9E+09]];
    CONST robtarget T961:=[[80.000004,52.487312,12.500005],[0.000000,0.000000,1.000000,0.000000],[0,0,-1,0],[9E+09,9E+09,9E+09,9E+09,9E+09,9E+09]];
    CONST robtarget T962:=[[80.000004,37.512688,12.500005],[0.000000,0.000000,1.000000,0.000000],[0,0,-1,0],[9E+09,9E+09,9E+09,9E+09,9E+09,9E+09]];
    CONST robtarget T963:=[[80.000004,30.000000,12.500005],[0.000000,0.000000,1.000000,0.000000],[0,0,-1,0],[9E+09,9E+09,9E+09,9E+09,9E+09,9E+09]];
    CONST robtarget T964:=[[78.739999,30.028279,12.500005],[0.000000,0.000000,1.000000,0.000000],[0,0,-1,0],[9E+09,9E+09,9E+09,9E+09,9E+09,9E+09]];
    CONST robtarget T965:=[[78.739999,37.608991,12.500005],[0.000000,0.000000,1.000000,0.000000],[0,0,-1,0],[9E+09,9E+09,9E+09,9E+09,9E+09,9E+09]];
    CONST robtarget T966:=[[78.739999,52.391011,12.500005],[0.000000,0.000000,1.000000,0.000000],[0,0,-1,0],[9E+09,9E+09,9E+09,9E+09,9E+09,9E+09]];
    CONST robtarget T967:=[[78.739999,72.608994,12.500005],[0.000000,0.000000,1.000000,0.000000],[0,0,-1,0],[9E+09,9E+09,9E+09,9E+09,9E+09,9E+09]];
    CONST robtarget T968:=[[78.739999,87.391014,12.500005],[0.000000,0.000000,1.000000,0.000000],[0,0,-1,0],[9E+09,9E+09,9E+09,9E+09,9E+09,9E+09]];
    CONST robtarget T969:=[[78.739999,107.608996,12.500005],[0.000000,0.000000,1.000000,0.000000],[0,0,-1,0],[9E+09,9E+09,9E+09,9E+09,9E+09,9E+09]];
    CONST robtarget T970:=[[78.739999,122.391017,12.500005],[0.000000,0.000000,1.000000,0.000000],[0,0,-1,0],[9E+09,9E+09,9E+09,9E+09,9E+09,9E+09]];
    CONST robtarget T971:=[[78.739999,129.971729,12.500005],[0.000000,0.000000,1.000000,0.000000],[0,0,-1,0],[9E+09,9E+09,9E+09,9E+09,9E+09,9E+09]];
    CONST robtarget T972:=[[77.479995,129.931001,12.500005],[0.000000,0.000000,1.000000,0.000000],[0,0,-1,0],[9E+09,9E+09,9E+09,9E+09,9E+09,9E+09]];
    CONST robtarget T973:=[[77.479995,122.050628,12.500005],[0.000000,0.000000,1.000000,0.000000],[0,0,-1,0],[9E+09,9E+09,9E+09,9E+09,9E+09,9E+09]];
    CONST robtarget T974:=[[77.479995,107.949384,12.500005],[0.000000,0.000000,1.000000,0.000000],[0,0,-1,0],[9E+09,9E+09,9E+09,9E+09,9E+09,9E+09]];
    CONST robtarget T975:=[[77.479995,87.050626,12.500005],[0.000000,0.000000,1.000000,0.000000],[0,0,-1,0],[9E+09,9E+09,9E+09,9E+09,9E+09,9E+09]];
    CONST robtarget T976:=[[77.479995,72.949381,12.500005],[0.000000,0.000000,1.000000,0.000000],[0,0,-1,0],[9E+09,9E+09,9E+09,9E+09,9E+09,9E+09]];
    CONST robtarget T977:=[[77.479995,52.050624,12.500005],[0.000000,0.000000,1.000000,0.000000],[0,0,-1,0],[9E+09,9E+09,9E+09,9E+09,9E+09,9E+09]];
    CONST robtarget T978:=[[77.479995,37.949379,12.500005],[0.000000,0.000000,1.000000,0.000000],[0,0,-1,0],[9E+09,9E+09,9E+09,9E+09,9E+09,9E+09]];
    CONST robtarget T979:=[[77.479995,30.069007,12.500005],[0.000000,0.000000,1.000000,0.000000],[0,0,-1,0],[9E+09,9E+09,9E+09,9E+09,9E+09,9E+09]];
    CONST robtarget T980:=[[76.219990,30.153959,12.500005],[0.000000,0.000000,1.000000,0.000000],[0,0,-1,0],[9E+09,9E+09,9E+09,9E+09,9E+09,9E+09]];
    CONST robtarget T981:=[[76.219990,38.524551,12.500005],[0.000000,0.000000,1.000000,0.000000],[0,0,-1,0],[9E+09,9E+09,9E+09,9E+09,9E+09,9E+09]];
    CONST robtarget T982:=[[76.219990,51.475451,12.500005],[0.000000,0.000000,1.000000,0.000000],[0,0,-1,0],[9E+09,9E+09,9E+09,9E+09,9E+09,9E+09]];
    CONST robtarget T983:=[[76.219990,73.524553,12.500005],[0.000000,0.000000,1.000000,0.000000],[0,0,-1,0],[9E+09,9E+09,9E+09,9E+09,9E+09,9E+09]];
    CONST robtarget T984:=[[76.219990,86.475455,12.500005],[0.000000,0.000000,1.000000,0.000000],[0,0,-1,0],[9E+09,9E+09,9E+09,9E+09,9E+09,9E+09]];
    CONST robtarget T985:=[[76.219990,108.524556,12.500005],[0.000000,0.000000,1.000000,0.000000],[0,0,-1,0],[9E+09,9E+09,9E+09,9E+09,9E+09,9E+09]];
    CONST robtarget T986:=[[76.219990,121.475457,12.500005],[0.000000,0.000000,1.000000,0.000000],[0,0,-1,0],[9E+09,9E+09,9E+09,9E+09,9E+09,9E+09]];
    CONST robtarget T987:=[[76.219990,129.846049,12.500005],[0.000000,0.000000,1.000000,0.000000],[0,0,-1,0],[9E+09,9E+09,9E+09,9E+09,9E+09,9E+09]];
    CONST robtarget T988:=[[74.959986,129.735844,12.500005],[0.000000,0.000000,1.000000,0.000000],[0,0,-1,0],[9E+09,9E+09,9E+09,9E+09,9E+09,9E+09]];
    CONST robtarget T989:=[[74.959986,120.544921,12.500005],[0.000000,0.000000,1.000000,0.000000],[0,0,-1,0],[9E+09,9E+09,9E+09,9E+09,9E+09,9E+09]];
    CONST robtarget T990:=[[74.959986,109.455091,12.500005],[0.000000,0.000000,1.000000,0.000000],[0,0,-1,0],[9E+09,9E+09,9E+09,9E+09,9E+09,9E+09]];
    CONST robtarget T991:=[[74.959986,85.544918,12.500005],[0.000000,0.000000,1.000000,0.000000],[0,0,-1,0],[9E+09,9E+09,9E+09,9E+09,9E+09,9E+09]];
    CONST robtarget T992:=[[74.959986,74.455090,12.500005],[0.000000,0.000000,1.000000,0.000000],[0,0,-1,0],[9E+09,9E+09,9E+09,9E+09,9E+09,9E+09]];
    CONST robtarget T993:=[[74.959986,50.544916,12.500005],[0.000000,0.000000,1.000000,0.000000],[0,0,-1,0],[9E+09,9E+09,9E+09,9E+09,9E+09,9E+09]];
    CONST robtarget T994:=[[74.959986,39.455086,12.500005],[0.000000,0.000000,1.000000,0.000000],[0,0,-1,0],[9E+09,9E+09,9E+09,9E+09,9E+09,9E+09]];
    CONST robtarget T995:=[[74.959986,30.264163,12.500005],[0.000000,0.000000,1.000000,0.000000],[0,0,-1,0],[9E+09,9E+09,9E+09,9E+09,9E+09,9E+09]];
    CONST robtarget T996:=[[73.699981,30.406130,12.500005],[0.000000,0.000000,1.000000,0.000000],[0,0,-1,0],[9E+09,9E+09,9E+09,9E+09,9E+09,9E+09]];
    CONST robtarget T997:=[[73.699981,40.937335,12.500005],[0.000000,0.000000,1.000000,0.000000],[0,0,-1,0],[9E+09,9E+09,9E+09,9E+09,9E+09,9E+09]];
    CONST robtarget T998:=[[73.699981,49.062665,12.500005],[0.000000,0.000000,1.000000,0.000000],[0,0,-1,0],[9E+09,9E+09,9E+09,9E+09,9E+09,9E+09]];
    CONST robtarget T999:=[[73.699981,75.937339,12.500005],[0.000000,0.000000,1.000000,0.000000],[0,0,-1,0],[9E+09,9E+09,9E+09,9E+09,9E+09,9E+09]];
    CONST robtarget T1000:=[[73.699981,84.062668,12.500005],[0.000000,0.000000,1.000000,0.000000],[0,0,-1,0],[9E+09,9E+09,9E+09,9E+09,9E+09,9E+09]];
    CONST robtarget T1001:=[[73.699981,110.937342,12.500005],[0.000000,0.000000,1.000000,0.000000],[0,0,-1,0],[9E+09,9E+09,9E+09,9E+09,9E+09,9E+09]];
    CONST robtarget T1002:=[[73.699981,119.062672,12.500005],[0.000000,0.000000,1.000000,0.000000],[0,0,-1,0],[9E+09,9E+09,9E+09,9E+09,9E+09,9E+09]];
    CONST robtarget T1003:=[[73.699981,129.593877,12.500005],[0.000000,0.000000,1.000000,0.000000],[0,0,-1,0],[9E+09,9E+09,9E+09,9E+09,9E+09,9E+09]];
    CONST robtarget T1004:=[[72.439977,129.413129,12.500005],[0.000000,0.000000,1.000000,0.000000],[0,0,-1,0],[9E+09,9E+09,9E+09,9E+09,9E+09,9E+09]];
    CONST robtarget T1005:=[[72.439977,30.586879,12.500005],[0.000000,0.000000,1.000000,0.000000],[0,0,-1,0],[9E+09,9E+09,9E+09,9E+09,9E+09,9E+09]];
    CONST robtarget T1006:=[[71.179972,30.786444,12.500005],[0.000000,0.000000,1.000000,0.000000],[0,0,-1,0],[9E+09,9E+09,9E+09,9E+09,9E+09,9E+09]];
    CONST robtarget T1007:=[[71.179972,129.213563,12.500005],[0.000000,0.000000,1.000000,0.000000],[0,0,-1,0],[9E+09,9E+09,9E+09,9E+09,9E+09,9E+09]];
    CONST robtarget T1008:=[[69.919968,128.960575,12.500005],[0.000000,0.000000,1.000000,0.000000],[0,0,-1,0],[9E+09,9E+09,9E+09,9E+09,9E+09,9E+09]];
    CONST robtarget T1009:=[[69.919968,31.039433,12.500005],[0.000000,0.000000,1.000000,0.000000],[0,0,-1,0],[9E+09,9E+09,9E+09,9E+09,9E+09,9E+09]];
    CONST robtarget T1010:=[[68.659963,31.307526,12.500005],[0.000000,0.000000,1.000000,0.000000],[0,0,-1,0],[9E+09,9E+09,9E+09,9E+09,9E+09,9E+09]];
    CONST robtarget T1011:=[[68.659963,128.692481,12.500005],[0.000000,0.000000,1.000000,0.000000],[0,0,-1,0],[9E+09,9E+09,9E+09,9E+09,9E+09,9E+09]];
    CONST robtarget T1012:=[[67.399959,128.374988,12.500005],[0.000000,0.000000,1.000000,0.000000],[0,0,-1,0],[9E+09,9E+09,9E+09,9E+09,9E+09,9E+09]];
    CONST robtarget T1013:=[[67.399959,31.625019,12.500005],[0.000000,0.000000,1.000000,0.000000],[0,0,-1,0],[9E+09,9E+09,9E+09,9E+09,9E+09,9E+09]];
    CONST robtarget T1014:=[[66.139954,31.969479,12.500005],[0.000000,0.000000,1.000000,0.000000],[0,0,-1,0],[9E+09,9E+09,9E+09,9E+09,9E+09,9E+09]];
    CONST robtarget T1015:=[[66.139954,128.030529,12.500005],[0.000000,0.000000,1.000000,0.000000],[0,0,-1,0],[9E+09,9E+09,9E+09,9E+09,9E+09,9E+09]];
    CONST robtarget T1016:=[[64.879950,127.652167,12.500005],[0.000000,0.000000,1.000000,0.000000],[0,0,-1,0],[9E+09,9E+09,9E+09,9E+09,9E+09,9E+09]];
    CONST robtarget T1017:=[[64.879950,32.347841,12.500005],[0.000000,0.000000,1.000000,0.000000],[0,0,-1,0],[9E+09,9E+09,9E+09,9E+09,9E+09,9E+09]];
    CONST robtarget T1018:=[[63.619945,32.772318,12.500005],[0.000000,0.000000,1.000000,0.000000],[0,0,-1,0],[9E+09,9E+09,9E+09,9E+09,9E+09,9E+09]];
    CONST robtarget T1019:=[[63.619945,127.227690,12.500005],[0.000000,0.000000,1.000000,0.000000],[0,0,-1,0],[9E+09,9E+09,9E+09,9E+09,9E+09,9E+09]];
    CONST robtarget T1020:=[[62.359941,126.783143,12.500005],[0.000000,0.000000,1.000000,0.000000],[0,0,-1,0],[9E+09,9E+09,9E+09,9E+09,9E+09,9E+09]];
    CONST robtarget T1021:=[[62.359941,33.216864,12.500005],[0.000000,0.000000,1.000000,0.000000],[0,0,-1,0],[9E+09,9E+09,9E+09,9E+09,9E+09,9E+09]];
    CONST robtarget T1022:=[[61.099936,33.722290,12.500005],[0.000000,0.000000,1.000000,0.000000],[0,0,-1,0],[9E+09,9E+09,9E+09,9E+09,9E+09,9E+09]];
    CONST robtarget T1023:=[[61.099936,126.277717,12.500005],[0.000000,0.000000,1.000000,0.000000],[0,0,-1,0],[9E+09,9E+09,9E+09,9E+09,9E+09,9E+09]];
    CONST robtarget T1024:=[[59.839932,125.745278,12.500005],[0.000000,0.000000,1.000000,0.000000],[0,0,-1,0],[9E+09,9E+09,9E+09,9E+09,9E+09,9E+09]];
    CONST robtarget T1025:=[[59.839932,34.254730,12.500005],[0.000000,0.000000,1.000000,0.000000],[0,0,-1,0],[9E+09,9E+09,9E+09,9E+09,9E+09,9E+09]];
    CONST robtarget T1026:=[[58.579927,34.827050,12.500005],[0.000000,0.000000,1.000000,0.000000],[0,0,-1,0],[9E+09,9E+09,9E+09,9E+09,9E+09,9E+09]];
    CONST robtarget T1027:=[[58.579927,125.172958,12.500005],[0.000000,0.000000,1.000000,0.000000],[0,0,-1,0],[9E+09,9E+09,9E+09,9E+09,9E+09,9E+09]];
    CONST robtarget T1028:=[[57.319923,124.546114,12.500005],[0.000000,0.000000,1.000000,0.000000],[0,0,-1,0],[9E+09,9E+09,9E+09,9E+09,9E+09,9E+09]];
    CONST robtarget T1029:=[[57.319923,35.453894,12.500005],[0.000000,0.000000,1.000000,0.000000],[0,0,-1,0],[9E+09,9E+09,9E+09,9E+09,9E+09,9E+09]];
    CONST robtarget T1030:=[[56.059918,36.110177,12.500005],[0.000000,0.000000,1.000000,0.000000],[0,0,-1,0],[9E+09,9E+09,9E+09,9E+09,9E+09,9E+09]];
    CONST robtarget T1031:=[[56.059918,123.889831,12.500005],[0.000000,0.000000,1.000000,0.000000],[0,0,-1,0],[9E+09,9E+09,9E+09,9E+09,9E+09,9E+09]];
    CONST robtarget T1032:=[[54.799914,123.174878,12.500005],[0.000000,0.000000,1.000000,0.000000],[0,0,-1,0],[9E+09,9E+09,9E+09,9E+09,9E+09,9E+09]];
    CONST robtarget T1033:=[[54.799914,36.825129,12.500005],[0.000000,0.000000,1.000000,0.000000],[0,0,-1,0],[9E+09,9E+09,9E+09,9E+09,9E+09,9E+09]];
    CONST robtarget T1034:=[[53.539909,37.589739,12.500005],[0.000000,0.000000,1.000000,0.000000],[0,0,-1,0],[9E+09,9E+09,9E+09,9E+09,9E+09,9E+09]];
    CONST robtarget T1035:=[[53.539909,122.410268,12.500005],[0.000000,0.000000,1.000000,0.000000],[0,0,-1,0],[9E+09,9E+09,9E+09,9E+09,9E+09,9E+09]];
    CONST robtarget T1036:=[[52.279905,121.607260,12.500005],[0.000000,0.000000,1.000000,0.000000],[0,0,-1,0],[9E+09,9E+09,9E+09,9E+09,9E+09,9E+09]];
    CONST robtarget T1037:=[[52.279905,81.789524,12.500005],[0.000000,0.000000,1.000000,0.000000],[0,0,-1,0],[9E+09,9E+09,9E+09,9E+09,9E+09,9E+09]];
    CONST robtarget T1038:=[[52.279905,78.210483,12.500005],[0.000000,0.000000,1.000000,0.000000],[0,0,-1,0],[9E+09,9E+09,9E+09,9E+09,9E+09,9E+09]];
    CONST robtarget T1039:=[[52.279905,38.392748,12.500005],[0.000000,0.000000,1.000000,0.000000],[0,0,-1,0],[9E+09,9E+09,9E+09,9E+09,9E+09,9E+09]];
    CONST robtarget T1040:=[[51.019900,39.265681,12.500005],[0.000000,0.000000,1.000000,0.000000],[0,0,-1,0],[9E+09,9E+09,9E+09,9E+09,9E+09,9E+09]];
    CONST robtarget T1041:=[[51.019900,75.547902,12.500005],[0.000000,0.000000,1.000000,0.000000],[0,0,-1,0],[9E+09,9E+09,9E+09,9E+09,9E+09,9E+09]];
    CONST robtarget T1042:=[[51.019900,84.452106,12.500005],[0.000000,0.000000,1.000000,0.000000],[0,0,-1,0],[9E+09,9E+09,9E+09,9E+09,9E+09,9E+09]];
    CONST robtarget T1043:=[[51.019900,120.734326,12.500005],[0.000000,0.000000,1.000000,0.000000],[0,0,-1,0],[9E+09,9E+09,9E+09,9E+09,9E+09,9E+09]];
    CONST robtarget T1044:=[[49.759896,119.803025,12.500005],[0.000000,0.000000,1.000000,0.000000],[0,0,-1,0],[9E+09,9E+09,9E+09,9E+09,9E+09,9E+09]];
    CONST robtarget T1045:=[[49.759896,85.779969,12.500005],[0.000000,0.000000,1.000000,0.000000],[0,0,-1,0],[9E+09,9E+09,9E+09,9E+09,9E+09,9E+09]];
    CONST robtarget T1046:=[[49.759896,74.220038,12.500005],[0.000000,0.000000,1.000000,0.000000],[0,0,-1,0],[9E+09,9E+09,9E+09,9E+09,9E+09,9E+09]];
    CONST robtarget T1047:=[[49.759896,40.196983,12.500005],[0.000000,0.000000,1.000000,0.000000],[0,0,-1,0],[9E+09,9E+09,9E+09,9E+09,9E+09,9E+09]];
    CONST robtarget T1048:=[[48.499891,41.180273,12.500005],[0.000000,0.000000,1.000000,0.000000],[0,0,-1,0],[9E+09,9E+09,9E+09,9E+09,9E+09,9E+09]];
    CONST robtarget T1049:=[[48.499891,73.379202,12.500005],[0.000000,0.000000,1.000000,0.000000],[0,0,-1,0],[9E+09,9E+09,9E+09,9E+09,9E+09,9E+09]];
    CONST robtarget T1050:=[[48.499891,86.620805,12.500005],[0.000000,0.000000,1.000000,0.000000],[0,0,-1,0],[9E+09,9E+09,9E+09,9E+09,9E+09,9E+09]];
    CONST robtarget T1051:=[[48.499891,118.819735,12.500005],[0.000000,0.000000,1.000000,0.000000],[0,0,-1,0],[9E+09,9E+09,9E+09,9E+09,9E+09,9E+09]];
    CONST robtarget T1052:=[[47.239887,117.767805,12.500005],[0.000000,0.000000,1.000000,0.000000],[0,0,-1,0],[9E+09,9E+09,9E+09,9E+09,9E+09,9E+09]];
    CONST robtarget T1053:=[[47.239887,87.152583,12.500005],[0.000000,0.000000,1.000000,0.000000],[0,0,-1,0],[9E+09,9E+09,9E+09,9E+09,9E+09,9E+09]];
    CONST robtarget T1054:=[[47.239887,72.847425,12.500005],[0.000000,0.000000,1.000000,0.000000],[0,0,-1,0],[9E+09,9E+09,9E+09,9E+09,9E+09,9E+09]];
    CONST robtarget T1055:=[[47.239887,42.232203,12.500005],[0.000000,0.000000,1.000000,0.000000],[0,0,-1,0],[9E+09,9E+09,9E+09,9E+09,9E+09,9E+09]];
    CONST robtarget T1056:=[[45.979882,43.373063,12.500005],[0.000000,0.000000,1.000000,0.000000],[0,0,-1,0],[9E+09,9E+09,9E+09,9E+09,9E+09,9E+09]];
    CONST robtarget T1057:=[[45.979882,72.576253,12.500005],[0.000000,0.000000,1.000000,0.000000],[0,0,-1,0],[9E+09,9E+09,9E+09,9E+09,9E+09,9E+09]];
    CONST robtarget T1058:=[[45.979882,87.423755,12.500005],[0.000000,0.000000,1.000000,0.000000],[0,0,-1,0],[9E+09,9E+09,9E+09,9E+09,9E+09,9E+09]];
    CONST robtarget T1059:=[[45.979882,116.626944,12.500005],[0.000000,0.000000,1.000000,0.000000],[0,0,-1,0],[9E+09,9E+09,9E+09,9E+09,9E+09,9E+09]];
    CONST robtarget T1060:=[[44.719878,115.412758,12.500005],[0.000000,0.000000,1.000000,0.000000],[0,0,-1,0],[9E+09,9E+09,9E+09,9E+09,9E+09,9E+09]];
    CONST robtarget T1061:=[[44.719878,87.487316,12.500005],[0.000000,0.000000,1.000000,0.000000],[0,0,-1,0],[9E+09,9E+09,9E+09,9E+09,9E+09,9E+09]];
    CONST robtarget T1062:=[[44.719878,72.512692,12.500005],[0.000000,0.000000,1.000000,0.000000],[0,0,-1,0],[9E+09,9E+09,9E+09,9E+09,9E+09,9E+09]];
    CONST robtarget T1063:=[[44.719878,44.587250,12.500005],[0.000000,0.000000,1.000000,0.000000],[0,0,-1,0],[9E+09,9E+09,9E+09,9E+09,9E+09,9E+09]];
    CONST robtarget T1064:=[[43.459873,45.884908,12.500005],[0.000000,0.000000,1.000000,0.000000],[0,0,-1,0],[9E+09,9E+09,9E+09,9E+09,9E+09,9E+09]];
    CONST robtarget T1065:=[[43.459873,72.670297,12.500005],[0.000000,0.000000,1.000000,0.000000],[0,0,-1,0],[9E+09,9E+09,9E+09,9E+09,9E+09,9E+09]];
    CONST robtarget T1066:=[[43.459873,87.329711,12.500005],[0.000000,0.000000,1.000000,0.000000],[0,0,-1,0],[9E+09,9E+09,9E+09,9E+09,9E+09,9E+09]];
    CONST robtarget T1067:=[[43.459873,114.115099,12.500005],[0.000000,0.000000,1.000000,0.000000],[0,0,-1,0],[9E+09,9E+09,9E+09,9E+09,9E+09,9E+09]];
    CONST robtarget T1068:=[[42.199869,112.721391,12.500005],[0.000000,0.000000,1.000000,0.000000],[0,0,-1,0],[9E+09,9E+09,9E+09,9E+09,9E+09,9E+09]];
    CONST robtarget T1069:=[[42.199869,86.948670,12.500005],[0.000000,0.000000,1.000000,0.000000],[0,0,-1,0],[9E+09,9E+09,9E+09,9E+09,9E+09,9E+09]];
    CONST robtarget T1070:=[[42.199869,73.051337,12.500005],[0.000000,0.000000,1.000000,0.000000],[0,0,-1,0],[9E+09,9E+09,9E+09,9E+09,9E+09,9E+09]];
    CONST robtarget T1071:=[[42.199869,47.278617,12.500005],[0.000000,0.000000,1.000000,0.000000],[0,0,-1,0],[9E+09,9E+09,9E+09,9E+09,9E+09,9E+09]];
    CONST robtarget T1072:=[[40.939864,48.787854,12.500005],[0.000000,0.000000,1.000000,0.000000],[0,0,-1,0],[9E+09,9E+09,9E+09,9E+09,9E+09,9E+09]];
    CONST robtarget T1073:=[[40.939864,73.708792,12.500005],[0.000000,0.000000,1.000000,0.000000],[0,0,-1,0],[9E+09,9E+09,9E+09,9E+09,9E+09,9E+09]];
    CONST robtarget T1074:=[[40.939864,86.291215,12.500005],[0.000000,0.000000,1.000000,0.000000],[0,0,-1,0],[9E+09,9E+09,9E+09,9E+09,9E+09,9E+09]];
    CONST robtarget T1075:=[[40.939864,111.212154,12.500005],[0.000000,0.000000,1.000000,0.000000],[0,0,-1,0],[9E+09,9E+09,9E+09,9E+09,9E+09,9E+09]];
    CONST robtarget T1076:=[[39.679860,109.560940,12.500005],[0.000000,0.000000,1.000000,0.000000],[0,0,-1,0],[9E+09,9E+09,9E+09,9E+09,9E+09,9E+09]];
    CONST robtarget T1077:=[[39.679860,85.271589,12.500005],[0.000000,0.000000,1.000000,0.000000],[0,0,-1,0],[9E+09,9E+09,9E+09,9E+09,9E+09,9E+09]];
    CONST robtarget T1078:=[[39.679860,74.728418,12.500005],[0.000000,0.000000,1.000000,0.000000],[0,0,-1,0],[9E+09,9E+09,9E+09,9E+09,9E+09,9E+09]];
    CONST robtarget T1079:=[[39.679860,50.439068,12.500005],[0.000000,0.000000,1.000000,0.000000],[0,0,-1,0],[9E+09,9E+09,9E+09,9E+09,9E+09,9E+09]];
    CONST robtarget T1080:=[[38.419855,52.240778,12.500005],[0.000000,0.000000,1.000000,0.000000],[0,0,-1,0],[9E+09,9E+09,9E+09,9E+09,9E+09,9E+09]];
    CONST robtarget T1081:=[[38.419855,76.422528,12.500005],[0.000000,0.000000,1.000000,0.000000],[0,0,-1,0],[9E+09,9E+09,9E+09,9E+09,9E+09,9E+09]];
    CONST robtarget T1082:=[[38.419855,83.577479,12.500005],[0.000000,0.000000,1.000000,0.000000],[0,0,-1,0],[9E+09,9E+09,9E+09,9E+09,9E+09,9E+09]];
    CONST robtarget T1083:=[[38.419855,107.759230,12.500005],[0.000000,0.000000,1.000000,0.000000],[0,0,-1,0],[9E+09,9E+09,9E+09,9E+09,9E+09,9E+09]];
    CONST robtarget T1084:=[[37.159851,105.775934,12.500005],[0.000000,0.000000,1.000000,0.000000],[0,0,-1,0],[9E+09,9E+09,9E+09,9E+09,9E+09,9E+09]];
    CONST robtarget T1085:=[[37.159851,54.224074,12.500005],[0.000000,0.000000,1.000000,0.000000],[0,0,-1,0],[9E+09,9E+09,9E+09,9E+09,9E+09,9E+09]];
    CONST robtarget T1086:=[[35.899846,56.444690,12.500005],[0.000000,0.000000,1.000000,0.000000],[0,0,-1,0],[9E+09,9E+09,9E+09,9E+09,9E+09,9E+09]];
    CONST robtarget T1087:=[[35.899846,103.555317,12.500005],[0.000000,0.000000,1.000000,0.000000],[0,0,-1,0],[9E+09,9E+09,9E+09,9E+09,9E+09,9E+09]];
    CONST robtarget T1088:=[[34.639842,101.007928,12.500005],[0.000000,0.000000,1.000000,0.000000],[0,0,-1,0],[9E+09,9E+09,9E+09,9E+09,9E+09,9E+09]];
    CONST robtarget T1089:=[[34.639842,58.992080,12.500005],[0.000000,0.000000,1.000000,0.000000],[0,0,-1,0],[9E+09,9E+09,9E+09,9E+09,9E+09,9E+09]];
    CONST robtarget T1090:=[[33.379837,61.953657,12.500005],[0.000000,0.000000,1.000000,0.000000],[0,0,-1,0],[9E+09,9E+09,9E+09,9E+09,9E+09,9E+09]];
    CONST robtarget T1091:=[[33.379837,98.046351,12.500005],[0.000000,0.000000,1.000000,0.000000],[0,0,-1,0],[9E+09,9E+09,9E+09,9E+09,9E+09,9E+09]];
    CONST robtarget T1092:=[[32.119833,94.360756,12.500005],[0.000000,0.000000,1.000000,0.000000],[0,0,-1,0],[9E+09,9E+09,9E+09,9E+09,9E+09,9E+09]];
    CONST robtarget T1093:=[[32.119833,65.639251,12.500005],[0.000000,0.000000,1.000000,0.000000],[0,0,-1,0],[9E+09,9E+09,9E+09,9E+09,9E+09,9E+09]];
    CONST robtarget T1094:=[[30.859828,70.797151,12.500005],[0.000000,0.000000,1.000000,0.000000],[0,0,-1,0],[9E+09,9E+09,9E+09,9E+09,9E+09,9E+09]];
    CONST robtarget T1095:=[[30.859828,89.202857,12.500005],[0.000000,0.000000,1.000000,0.000000],[0,0,-1,0],[9E+09,9E+09,9E+09,9E+09,9E+09,9E+09]];
    CONST robtarget T1096:=[[30.859828,70.797151,13.200015],[0.000000,0.000000,1.000000,0.000000],[0,0,-1,0],[9E+09,9E+09,9E+09,9E+09,9E+09,9E+09]];
    CONST robtarget T1097:=[[30.859828,89.202857,13.200015],[0.000000,0.000000,1.000000,0.000000],[0,0,-1,0],[9E+09,9E+09,9E+09,9E+09,9E+09,9E+09]];
    CONST robtarget T1098:=[[30.859828,70.797151,13.200015],[0.000000,0.000000,1.000000,0.000000],[0,0,-1,0],[9E+09,9E+09,9E+09,9E+09,9E+09,9E+09]];
    CONST robtarget T1099:=[[30.859828,89.202857,13.200015],[0.000000,0.000000,1.000000,0.000000],[0,0,-1,0],[9E+09,9E+09,9E+09,9E+09,9E+09,9E+09]];
    CONST robtarget T1100:=[[32.119833,94.360756,13.200015],[0.000000,0.000000,1.000000,0.000000],[0,0,-1,0],[9E+09,9E+09,9E+09,9E+09,9E+09,9E+09]];
    CONST robtarget T1101:=[[32.119833,65.639251,13.200015],[0.000000,0.000000,1.000000,0.000000],[0,0,-1,0],[9E+09,9E+09,9E+09,9E+09,9E+09,9E+09]];
    CONST robtarget T1102:=[[33.379837,61.953657,13.200015],[0.000000,0.000000,1.000000,0.000000],[0,0,-1,0],[9E+09,9E+09,9E+09,9E+09,9E+09,9E+09]];
    CONST robtarget T1103:=[[33.379837,98.046351,13.200015],[0.000000,0.000000,1.000000,0.000000],[0,0,-1,0],[9E+09,9E+09,9E+09,9E+09,9E+09,9E+09]];
    CONST robtarget T1104:=[[34.639842,101.007928,13.200015],[0.000000,0.000000,1.000000,0.000000],[0,0,-1,0],[9E+09,9E+09,9E+09,9E+09,9E+09,9E+09]];
    CONST robtarget T1105:=[[34.639842,58.992080,13.200015],[0.000000,0.000000,1.000000,0.000000],[0,0,-1,0],[9E+09,9E+09,9E+09,9E+09,9E+09,9E+09]];
    CONST robtarget T1106:=[[35.899846,56.444690,13.200015],[0.000000,0.000000,1.000000,0.000000],[0,0,-1,0],[9E+09,9E+09,9E+09,9E+09,9E+09,9E+09]];
    CONST robtarget T1107:=[[35.899846,103.555317,13.200015],[0.000000,0.000000,1.000000,0.000000],[0,0,-1,0],[9E+09,9E+09,9E+09,9E+09,9E+09,9E+09]];
    CONST robtarget T1108:=[[37.159851,105.775934,13.200015],[0.000000,0.000000,1.000000,0.000000],[0,0,-1,0],[9E+09,9E+09,9E+09,9E+09,9E+09,9E+09]];
    CONST robtarget T1109:=[[37.159851,54.224074,13.200015],[0.000000,0.000000,1.000000,0.000000],[0,0,-1,0],[9E+09,9E+09,9E+09,9E+09,9E+09,9E+09]];
    CONST robtarget T1110:=[[38.419855,52.240778,13.200015],[0.000000,0.000000,1.000000,0.000000],[0,0,-1,0],[9E+09,9E+09,9E+09,9E+09,9E+09,9E+09]];
    CONST robtarget T1111:=[[38.419855,76.422528,13.200015],[0.000000,0.000000,1.000000,0.000000],[0,0,-1,0],[9E+09,9E+09,9E+09,9E+09,9E+09,9E+09]];
    CONST robtarget T1112:=[[38.419855,83.577479,13.200015],[0.000000,0.000000,1.000000,0.000000],[0,0,-1,0],[9E+09,9E+09,9E+09,9E+09,9E+09,9E+09]];
    CONST robtarget T1113:=[[38.419855,107.759230,13.200015],[0.000000,0.000000,1.000000,0.000000],[0,0,-1,0],[9E+09,9E+09,9E+09,9E+09,9E+09,9E+09]];
    CONST robtarget T1114:=[[39.679860,109.560940,13.200015],[0.000000,0.000000,1.000000,0.000000],[0,0,-1,0],[9E+09,9E+09,9E+09,9E+09,9E+09,9E+09]];
    CONST robtarget T1115:=[[39.679860,85.271589,13.200015],[0.000000,0.000000,1.000000,0.000000],[0,0,-1,0],[9E+09,9E+09,9E+09,9E+09,9E+09,9E+09]];
    CONST robtarget T1116:=[[39.679860,74.728418,13.200015],[0.000000,0.000000,1.000000,0.000000],[0,0,-1,0],[9E+09,9E+09,9E+09,9E+09,9E+09,9E+09]];
    CONST robtarget T1117:=[[39.679860,50.439068,13.200015],[0.000000,0.000000,1.000000,0.000000],[0,0,-1,0],[9E+09,9E+09,9E+09,9E+09,9E+09,9E+09]];
    CONST robtarget T1118:=[[40.939864,48.787854,13.200015],[0.000000,0.000000,1.000000,0.000000],[0,0,-1,0],[9E+09,9E+09,9E+09,9E+09,9E+09,9E+09]];
    CONST robtarget T1119:=[[40.939864,73.708792,13.200015],[0.000000,0.000000,1.000000,0.000000],[0,0,-1,0],[9E+09,9E+09,9E+09,9E+09,9E+09,9E+09]];
    CONST robtarget T1120:=[[40.939864,86.291215,13.200015],[0.000000,0.000000,1.000000,0.000000],[0,0,-1,0],[9E+09,9E+09,9E+09,9E+09,9E+09,9E+09]];
    CONST robtarget T1121:=[[40.939864,111.212154,13.200015],[0.000000,0.000000,1.000000,0.000000],[0,0,-1,0],[9E+09,9E+09,9E+09,9E+09,9E+09,9E+09]];
    CONST robtarget T1122:=[[42.199869,112.721391,13.200015],[0.000000,0.000000,1.000000,0.000000],[0,0,-1,0],[9E+09,9E+09,9E+09,9E+09,9E+09,9E+09]];
    CONST robtarget T1123:=[[42.199869,86.948670,13.200015],[0.000000,0.000000,1.000000,0.000000],[0,0,-1,0],[9E+09,9E+09,9E+09,9E+09,9E+09,9E+09]];
    CONST robtarget T1124:=[[42.199869,73.051337,13.200015],[0.000000,0.000000,1.000000,0.000000],[0,0,-1,0],[9E+09,9E+09,9E+09,9E+09,9E+09,9E+09]];
    CONST robtarget T1125:=[[42.199869,47.278617,13.200015],[0.000000,0.000000,1.000000,0.000000],[0,0,-1,0],[9E+09,9E+09,9E+09,9E+09,9E+09,9E+09]];
    CONST robtarget T1126:=[[43.459873,45.884908,13.200015],[0.000000,0.000000,1.000000,0.000000],[0,0,-1,0],[9E+09,9E+09,9E+09,9E+09,9E+09,9E+09]];
    CONST robtarget T1127:=[[43.459873,72.670297,13.200015],[0.000000,0.000000,1.000000,0.000000],[0,0,-1,0],[9E+09,9E+09,9E+09,9E+09,9E+09,9E+09]];
    CONST robtarget T1128:=[[43.459873,87.329711,13.200015],[0.000000,0.000000,1.000000,0.000000],[0,0,-1,0],[9E+09,9E+09,9E+09,9E+09,9E+09,9E+09]];
    CONST robtarget T1129:=[[43.459873,114.115099,13.200015],[0.000000,0.000000,1.000000,0.000000],[0,0,-1,0],[9E+09,9E+09,9E+09,9E+09,9E+09,9E+09]];
    CONST robtarget T1130:=[[44.719878,115.412758,13.200015],[0.000000,0.000000,1.000000,0.000000],[0,0,-1,0],[9E+09,9E+09,9E+09,9E+09,9E+09,9E+09]];
    CONST robtarget T1131:=[[44.719878,87.487316,13.200015],[0.000000,0.000000,1.000000,0.000000],[0,0,-1,0],[9E+09,9E+09,9E+09,9E+09,9E+09,9E+09]];
    CONST robtarget T1132:=[[44.719878,72.512692,13.200015],[0.000000,0.000000,1.000000,0.000000],[0,0,-1,0],[9E+09,9E+09,9E+09,9E+09,9E+09,9E+09]];
    CONST robtarget T1133:=[[44.719878,44.587250,13.200015],[0.000000,0.000000,1.000000,0.000000],[0,0,-1,0],[9E+09,9E+09,9E+09,9E+09,9E+09,9E+09]];
    CONST robtarget T1134:=[[45.979882,43.373063,13.200015],[0.000000,0.000000,1.000000,0.000000],[0,0,-1,0],[9E+09,9E+09,9E+09,9E+09,9E+09,9E+09]];
    CONST robtarget T1135:=[[45.979882,72.576253,13.200015],[0.000000,0.000000,1.000000,0.000000],[0,0,-1,0],[9E+09,9E+09,9E+09,9E+09,9E+09,9E+09]];
    CONST robtarget T1136:=[[45.979882,87.423755,13.200015],[0.000000,0.000000,1.000000,0.000000],[0,0,-1,0],[9E+09,9E+09,9E+09,9E+09,9E+09,9E+09]];
    CONST robtarget T1137:=[[45.979882,116.626944,13.200015],[0.000000,0.000000,1.000000,0.000000],[0,0,-1,0],[9E+09,9E+09,9E+09,9E+09,9E+09,9E+09]];
    CONST robtarget T1138:=[[47.239887,117.767805,13.200015],[0.000000,0.000000,1.000000,0.000000],[0,0,-1,0],[9E+09,9E+09,9E+09,9E+09,9E+09,9E+09]];
    CONST robtarget T1139:=[[47.239887,87.152583,13.200015],[0.000000,0.000000,1.000000,0.000000],[0,0,-1,0],[9E+09,9E+09,9E+09,9E+09,9E+09,9E+09]];
    CONST robtarget T1140:=[[47.239887,72.847425,13.200015],[0.000000,0.000000,1.000000,0.000000],[0,0,-1,0],[9E+09,9E+09,9E+09,9E+09,9E+09,9E+09]];
    CONST robtarget T1141:=[[47.239887,42.232203,13.200015],[0.000000,0.000000,1.000000,0.000000],[0,0,-1,0],[9E+09,9E+09,9E+09,9E+09,9E+09,9E+09]];
    CONST robtarget T1142:=[[48.499891,41.180273,13.200015],[0.000000,0.000000,1.000000,0.000000],[0,0,-1,0],[9E+09,9E+09,9E+09,9E+09,9E+09,9E+09]];
    CONST robtarget T1143:=[[48.499891,73.379202,13.200015],[0.000000,0.000000,1.000000,0.000000],[0,0,-1,0],[9E+09,9E+09,9E+09,9E+09,9E+09,9E+09]];
    CONST robtarget T1144:=[[48.499891,86.620805,13.200015],[0.000000,0.000000,1.000000,0.000000],[0,0,-1,0],[9E+09,9E+09,9E+09,9E+09,9E+09,9E+09]];
    CONST robtarget T1145:=[[48.499891,118.819735,13.200015],[0.000000,0.000000,1.000000,0.000000],[0,0,-1,0],[9E+09,9E+09,9E+09,9E+09,9E+09,9E+09]];
    CONST robtarget T1146:=[[49.759896,119.803025,13.200015],[0.000000,0.000000,1.000000,0.000000],[0,0,-1,0],[9E+09,9E+09,9E+09,9E+09,9E+09,9E+09]];
    CONST robtarget T1147:=[[49.759896,85.779969,13.200015],[0.000000,0.000000,1.000000,0.000000],[0,0,-1,0],[9E+09,9E+09,9E+09,9E+09,9E+09,9E+09]];
    CONST robtarget T1148:=[[49.759896,74.220038,13.200015],[0.000000,0.000000,1.000000,0.000000],[0,0,-1,0],[9E+09,9E+09,9E+09,9E+09,9E+09,9E+09]];
    CONST robtarget T1149:=[[49.759896,40.196983,13.200015],[0.000000,0.000000,1.000000,0.000000],[0,0,-1,0],[9E+09,9E+09,9E+09,9E+09,9E+09,9E+09]];
    CONST robtarget T1150:=[[51.019900,39.265681,13.200015],[0.000000,0.000000,1.000000,0.000000],[0,0,-1,0],[9E+09,9E+09,9E+09,9E+09,9E+09,9E+09]];
    CONST robtarget T1151:=[[51.019900,75.547902,13.200015],[0.000000,0.000000,1.000000,0.000000],[0,0,-1,0],[9E+09,9E+09,9E+09,9E+09,9E+09,9E+09]];
    CONST robtarget T1152:=[[51.019900,84.452106,13.200015],[0.000000,0.000000,1.000000,0.000000],[0,0,-1,0],[9E+09,9E+09,9E+09,9E+09,9E+09,9E+09]];
    CONST robtarget T1153:=[[51.019900,120.734326,13.200015],[0.000000,0.000000,1.000000,0.000000],[0,0,-1,0],[9E+09,9E+09,9E+09,9E+09,9E+09,9E+09]];
    CONST robtarget T1154:=[[52.279905,121.607260,13.200015],[0.000000,0.000000,1.000000,0.000000],[0,0,-1,0],[9E+09,9E+09,9E+09,9E+09,9E+09,9E+09]];
    CONST robtarget T1155:=[[52.279905,81.789524,13.200015],[0.000000,0.000000,1.000000,0.000000],[0,0,-1,0],[9E+09,9E+09,9E+09,9E+09,9E+09,9E+09]];
    CONST robtarget T1156:=[[52.279905,78.210483,13.200015],[0.000000,0.000000,1.000000,0.000000],[0,0,-1,0],[9E+09,9E+09,9E+09,9E+09,9E+09,9E+09]];
    CONST robtarget T1157:=[[52.279905,38.392748,13.200015],[0.000000,0.000000,1.000000,0.000000],[0,0,-1,0],[9E+09,9E+09,9E+09,9E+09,9E+09,9E+09]];
    CONST robtarget T1158:=[[53.539909,37.589739,13.200015],[0.000000,0.000000,1.000000,0.000000],[0,0,-1,0],[9E+09,9E+09,9E+09,9E+09,9E+09,9E+09]];
    CONST robtarget T1159:=[[53.539909,122.410268,13.200015],[0.000000,0.000000,1.000000,0.000000],[0,0,-1,0],[9E+09,9E+09,9E+09,9E+09,9E+09,9E+09]];
    CONST robtarget T1160:=[[54.799914,123.174878,13.200015],[0.000000,0.000000,1.000000,0.000000],[0,0,-1,0],[9E+09,9E+09,9E+09,9E+09,9E+09,9E+09]];
    CONST robtarget T1161:=[[54.799914,36.825129,13.200015],[0.000000,0.000000,1.000000,0.000000],[0,0,-1,0],[9E+09,9E+09,9E+09,9E+09,9E+09,9E+09]];
    CONST robtarget T1162:=[[56.059918,36.110177,13.200015],[0.000000,0.000000,1.000000,0.000000],[0,0,-1,0],[9E+09,9E+09,9E+09,9E+09,9E+09,9E+09]];
    CONST robtarget T1163:=[[56.059918,123.889831,13.200015],[0.000000,0.000000,1.000000,0.000000],[0,0,-1,0],[9E+09,9E+09,9E+09,9E+09,9E+09,9E+09]];
    CONST robtarget T1164:=[[57.319923,124.546114,13.200015],[0.000000,0.000000,1.000000,0.000000],[0,0,-1,0],[9E+09,9E+09,9E+09,9E+09,9E+09,9E+09]];
    CONST robtarget T1165:=[[57.319923,35.453894,13.200015],[0.000000,0.000000,1.000000,0.000000],[0,0,-1,0],[9E+09,9E+09,9E+09,9E+09,9E+09,9E+09]];
    CONST robtarget T1166:=[[58.579927,34.827050,13.200015],[0.000000,0.000000,1.000000,0.000000],[0,0,-1,0],[9E+09,9E+09,9E+09,9E+09,9E+09,9E+09]];
    CONST robtarget T1167:=[[58.579927,125.172958,13.200015],[0.000000,0.000000,1.000000,0.000000],[0,0,-1,0],[9E+09,9E+09,9E+09,9E+09,9E+09,9E+09]];
    CONST robtarget T1168:=[[59.839932,125.745278,13.200015],[0.000000,0.000000,1.000000,0.000000],[0,0,-1,0],[9E+09,9E+09,9E+09,9E+09,9E+09,9E+09]];
    CONST robtarget T1169:=[[59.839932,34.254730,13.200015],[0.000000,0.000000,1.000000,0.000000],[0,0,-1,0],[9E+09,9E+09,9E+09,9E+09,9E+09,9E+09]];
    CONST robtarget T1170:=[[61.099936,33.722290,13.200015],[0.000000,0.000000,1.000000,0.000000],[0,0,-1,0],[9E+09,9E+09,9E+09,9E+09,9E+09,9E+09]];
    CONST robtarget T1171:=[[61.099936,126.277717,13.200015],[0.000000,0.000000,1.000000,0.000000],[0,0,-1,0],[9E+09,9E+09,9E+09,9E+09,9E+09,9E+09]];
    CONST robtarget T1172:=[[62.359941,126.783143,13.200015],[0.000000,0.000000,1.000000,0.000000],[0,0,-1,0],[9E+09,9E+09,9E+09,9E+09,9E+09,9E+09]];
    CONST robtarget T1173:=[[62.359941,33.216864,13.200015],[0.000000,0.000000,1.000000,0.000000],[0,0,-1,0],[9E+09,9E+09,9E+09,9E+09,9E+09,9E+09]];
    CONST robtarget T1174:=[[63.619945,32.772318,13.200015],[0.000000,0.000000,1.000000,0.000000],[0,0,-1,0],[9E+09,9E+09,9E+09,9E+09,9E+09,9E+09]];
    CONST robtarget T1175:=[[63.619945,127.227690,13.200015],[0.000000,0.000000,1.000000,0.000000],[0,0,-1,0],[9E+09,9E+09,9E+09,9E+09,9E+09,9E+09]];
    CONST robtarget T1176:=[[64.879950,127.652167,13.200015],[0.000000,0.000000,1.000000,0.000000],[0,0,-1,0],[9E+09,9E+09,9E+09,9E+09,9E+09,9E+09]];
    CONST robtarget T1177:=[[64.879950,32.347841,13.200015],[0.000000,0.000000,1.000000,0.000000],[0,0,-1,0],[9E+09,9E+09,9E+09,9E+09,9E+09,9E+09]];
    CONST robtarget T1178:=[[66.139954,31.969479,13.200015],[0.000000,0.000000,1.000000,0.000000],[0,0,-1,0],[9E+09,9E+09,9E+09,9E+09,9E+09,9E+09]];
    CONST robtarget T1179:=[[66.139954,128.030529,13.200015],[0.000000,0.000000,1.000000,0.000000],[0,0,-1,0],[9E+09,9E+09,9E+09,9E+09,9E+09,9E+09]];
    CONST robtarget T1180:=[[67.399959,128.374988,13.200015],[0.000000,0.000000,1.000000,0.000000],[0,0,-1,0],[9E+09,9E+09,9E+09,9E+09,9E+09,9E+09]];
    CONST robtarget T1181:=[[67.399959,31.625019,13.200015],[0.000000,0.000000,1.000000,0.000000],[0,0,-1,0],[9E+09,9E+09,9E+09,9E+09,9E+09,9E+09]];
    CONST robtarget T1182:=[[68.659963,31.307526,13.200015],[0.000000,0.000000,1.000000,0.000000],[0,0,-1,0],[9E+09,9E+09,9E+09,9E+09,9E+09,9E+09]];
    CONST robtarget T1183:=[[68.659963,128.692481,13.200015],[0.000000,0.000000,1.000000,0.000000],[0,0,-1,0],[9E+09,9E+09,9E+09,9E+09,9E+09,9E+09]];
    CONST robtarget T1184:=[[69.919968,128.960575,13.200015],[0.000000,0.000000,1.000000,0.000000],[0,0,-1,0],[9E+09,9E+09,9E+09,9E+09,9E+09,9E+09]];
    CONST robtarget T1185:=[[69.919968,31.039433,13.200015],[0.000000,0.000000,1.000000,0.000000],[0,0,-1,0],[9E+09,9E+09,9E+09,9E+09,9E+09,9E+09]];
    CONST robtarget T1186:=[[71.179972,30.786444,13.200015],[0.000000,0.000000,1.000000,0.000000],[0,0,-1,0],[9E+09,9E+09,9E+09,9E+09,9E+09,9E+09]];
    CONST robtarget T1187:=[[71.179972,129.213563,13.200015],[0.000000,0.000000,1.000000,0.000000],[0,0,-1,0],[9E+09,9E+09,9E+09,9E+09,9E+09,9E+09]];
    CONST robtarget T1188:=[[72.439977,129.413129,13.200015],[0.000000,0.000000,1.000000,0.000000],[0,0,-1,0],[9E+09,9E+09,9E+09,9E+09,9E+09,9E+09]];
    CONST robtarget T1189:=[[72.439977,30.586879,13.200015],[0.000000,0.000000,1.000000,0.000000],[0,0,-1,0],[9E+09,9E+09,9E+09,9E+09,9E+09,9E+09]];
    CONST robtarget T1190:=[[73.699981,30.406130,13.200015],[0.000000,0.000000,1.000000,0.000000],[0,0,-1,0],[9E+09,9E+09,9E+09,9E+09,9E+09,9E+09]];
    CONST robtarget T1191:=[[73.699981,40.937335,13.200015],[0.000000,0.000000,1.000000,0.000000],[0,0,-1,0],[9E+09,9E+09,9E+09,9E+09,9E+09,9E+09]];
    CONST robtarget T1192:=[[73.699981,49.062665,13.200015],[0.000000,0.000000,1.000000,0.000000],[0,0,-1,0],[9E+09,9E+09,9E+09,9E+09,9E+09,9E+09]];
    CONST robtarget T1193:=[[73.699981,75.937339,13.200015],[0.000000,0.000000,1.000000,0.000000],[0,0,-1,0],[9E+09,9E+09,9E+09,9E+09,9E+09,9E+09]];
    CONST robtarget T1194:=[[73.699981,84.062668,13.200015],[0.000000,0.000000,1.000000,0.000000],[0,0,-1,0],[9E+09,9E+09,9E+09,9E+09,9E+09,9E+09]];
    CONST robtarget T1195:=[[73.699981,110.937342,13.200015],[0.000000,0.000000,1.000000,0.000000],[0,0,-1,0],[9E+09,9E+09,9E+09,9E+09,9E+09,9E+09]];
    CONST robtarget T1196:=[[73.699981,119.062672,13.200015],[0.000000,0.000000,1.000000,0.000000],[0,0,-1,0],[9E+09,9E+09,9E+09,9E+09,9E+09,9E+09]];
    CONST robtarget T1197:=[[73.699981,129.593877,13.200015],[0.000000,0.000000,1.000000,0.000000],[0,0,-1,0],[9E+09,9E+09,9E+09,9E+09,9E+09,9E+09]];
    CONST robtarget T1198:=[[74.959986,129.735844,13.200015],[0.000000,0.000000,1.000000,0.000000],[0,0,-1,0],[9E+09,9E+09,9E+09,9E+09,9E+09,9E+09]];
    CONST robtarget T1199:=[[74.959986,120.544921,13.200015],[0.000000,0.000000,1.000000,0.000000],[0,0,-1,0],[9E+09,9E+09,9E+09,9E+09,9E+09,9E+09]];
    CONST robtarget T1200:=[[74.959986,109.455091,13.200015],[0.000000,0.000000,1.000000,0.000000],[0,0,-1,0],[9E+09,9E+09,9E+09,9E+09,9E+09,9E+09]];
    CONST robtarget T1201:=[[74.959986,85.544918,13.200015],[0.000000,0.000000,1.000000,0.000000],[0,0,-1,0],[9E+09,9E+09,9E+09,9E+09,9E+09,9E+09]];
    CONST robtarget T1202:=[[74.959986,74.455090,13.200015],[0.000000,0.000000,1.000000,0.000000],[0,0,-1,0],[9E+09,9E+09,9E+09,9E+09,9E+09,9E+09]];
    CONST robtarget T1203:=[[74.959986,50.544916,13.200015],[0.000000,0.000000,1.000000,0.000000],[0,0,-1,0],[9E+09,9E+09,9E+09,9E+09,9E+09,9E+09]];
    CONST robtarget T1204:=[[74.959986,39.455086,13.200015],[0.000000,0.000000,1.000000,0.000000],[0,0,-1,0],[9E+09,9E+09,9E+09,9E+09,9E+09,9E+09]];
    CONST robtarget T1205:=[[74.959986,30.264163,13.200015],[0.000000,0.000000,1.000000,0.000000],[0,0,-1,0],[9E+09,9E+09,9E+09,9E+09,9E+09,9E+09]];
    CONST robtarget T1206:=[[76.219990,30.153959,13.200015],[0.000000,0.000000,1.000000,0.000000],[0,0,-1,0],[9E+09,9E+09,9E+09,9E+09,9E+09,9E+09]];
    CONST robtarget T1207:=[[76.219990,38.524551,13.200015],[0.000000,0.000000,1.000000,0.000000],[0,0,-1,0],[9E+09,9E+09,9E+09,9E+09,9E+09,9E+09]];
    CONST robtarget T1208:=[[76.219990,51.475451,13.200015],[0.000000,0.000000,1.000000,0.000000],[0,0,-1,0],[9E+09,9E+09,9E+09,9E+09,9E+09,9E+09]];
    CONST robtarget T1209:=[[76.219990,73.524553,13.200015],[0.000000,0.000000,1.000000,0.000000],[0,0,-1,0],[9E+09,9E+09,9E+09,9E+09,9E+09,9E+09]];
    CONST robtarget T1210:=[[76.219990,86.475455,13.200015],[0.000000,0.000000,1.000000,0.000000],[0,0,-1,0],[9E+09,9E+09,9E+09,9E+09,9E+09,9E+09]];
    CONST robtarget T1211:=[[76.219990,108.524556,13.200015],[0.000000,0.000000,1.000000,0.000000],[0,0,-1,0],[9E+09,9E+09,9E+09,9E+09,9E+09,9E+09]];
    CONST robtarget T1212:=[[76.219990,121.475457,13.200015],[0.000000,0.000000,1.000000,0.000000],[0,0,-1,0],[9E+09,9E+09,9E+09,9E+09,9E+09,9E+09]];
    CONST robtarget T1213:=[[76.219990,129.846049,13.200015],[0.000000,0.000000,1.000000,0.000000],[0,0,-1,0],[9E+09,9E+09,9E+09,9E+09,9E+09,9E+09]];
    CONST robtarget T1214:=[[77.479995,129.931001,13.200015],[0.000000,0.000000,1.000000,0.000000],[0,0,-1,0],[9E+09,9E+09,9E+09,9E+09,9E+09,9E+09]];
    CONST robtarget T1215:=[[77.479995,122.050628,13.200015],[0.000000,0.000000,1.000000,0.000000],[0,0,-1,0],[9E+09,9E+09,9E+09,9E+09,9E+09,9E+09]];
    CONST robtarget T1216:=[[77.479995,107.949384,13.200015],[0.000000,0.000000,1.000000,0.000000],[0,0,-1,0],[9E+09,9E+09,9E+09,9E+09,9E+09,9E+09]];
    CONST robtarget T1217:=[[77.479995,87.050626,13.200015],[0.000000,0.000000,1.000000,0.000000],[0,0,-1,0],[9E+09,9E+09,9E+09,9E+09,9E+09,9E+09]];
    CONST robtarget T1218:=[[77.479995,72.949381,13.200015],[0.000000,0.000000,1.000000,0.000000],[0,0,-1,0],[9E+09,9E+09,9E+09,9E+09,9E+09,9E+09]];
    CONST robtarget T1219:=[[77.479995,52.050624,13.200015],[0.000000,0.000000,1.000000,0.000000],[0,0,-1,0],[9E+09,9E+09,9E+09,9E+09,9E+09,9E+09]];
    CONST robtarget T1220:=[[77.479995,37.949379,13.200015],[0.000000,0.000000,1.000000,0.000000],[0,0,-1,0],[9E+09,9E+09,9E+09,9E+09,9E+09,9E+09]];
    CONST robtarget T1221:=[[77.479995,30.069007,13.200015],[0.000000,0.000000,1.000000,0.000000],[0,0,-1,0],[9E+09,9E+09,9E+09,9E+09,9E+09,9E+09]];
    CONST robtarget T1222:=[[78.739999,30.028279,13.200015],[0.000000,0.000000,1.000000,0.000000],[0,0,-1,0],[9E+09,9E+09,9E+09,9E+09,9E+09,9E+09]];
    CONST robtarget T1223:=[[78.739999,37.608991,13.200015],[0.000000,0.000000,1.000000,0.000000],[0,0,-1,0],[9E+09,9E+09,9E+09,9E+09,9E+09,9E+09]];
    CONST robtarget T1224:=[[78.739999,52.391011,13.200015],[0.000000,0.000000,1.000000,0.000000],[0,0,-1,0],[9E+09,9E+09,9E+09,9E+09,9E+09,9E+09]];
    CONST robtarget T1225:=[[78.739999,72.608994,13.200015],[0.000000,0.000000,1.000000,0.000000],[0,0,-1,0],[9E+09,9E+09,9E+09,9E+09,9E+09,9E+09]];
    CONST robtarget T1226:=[[78.739999,87.391014,13.200015],[0.000000,0.000000,1.000000,0.000000],[0,0,-1,0],[9E+09,9E+09,9E+09,9E+09,9E+09,9E+09]];
    CONST robtarget T1227:=[[78.739999,107.608996,13.200015],[0.000000,0.000000,1.000000,0.000000],[0,0,-1,0],[9E+09,9E+09,9E+09,9E+09,9E+09,9E+09]];
    CONST robtarget T1228:=[[78.739999,122.391017,13.200015],[0.000000,0.000000,1.000000,0.000000],[0,0,-1,0],[9E+09,9E+09,9E+09,9E+09,9E+09,9E+09]];
    CONST robtarget T1229:=[[78.739999,129.971729,13.200015],[0.000000,0.000000,1.000000,0.000000],[0,0,-1,0],[9E+09,9E+09,9E+09,9E+09,9E+09,9E+09]];
    CONST robtarget T1230:=[[80.000004,130.000008,13.200015],[0.000000,0.000000,1.000000,0.000000],[0,0,-1,0],[9E+09,9E+09,9E+09,9E+09,9E+09,9E+09]];
    CONST robtarget T1231:=[[80.000004,122.487319,13.200015],[0.000000,0.000000,1.000000,0.000000],[0,0,-1,0],[9E+09,9E+09,9E+09,9E+09,9E+09,9E+09]];
    CONST robtarget T1232:=[[80.000004,107.512696,13.200015],[0.000000,0.000000,1.000000,0.000000],[0,0,-1,0],[9E+09,9E+09,9E+09,9E+09,9E+09,9E+09]];
    CONST robtarget T1233:=[[80.000004,87.487316,13.200015],[0.000000,0.000000,1.000000,0.000000],[0,0,-1,0],[9E+09,9E+09,9E+09,9E+09,9E+09,9E+09]];
    CONST robtarget T1234:=[[80.000004,72.512692,13.200015],[0.000000,0.000000,1.000000,0.000000],[0,0,-1,0],[9E+09,9E+09,9E+09,9E+09,9E+09,9E+09]];
    CONST robtarget T1235:=[[80.000004,52.487312,13.200015],[0.000000,0.000000,1.000000,0.000000],[0,0,-1,0],[9E+09,9E+09,9E+09,9E+09,9E+09,9E+09]];
    CONST robtarget T1236:=[[80.000004,37.512688,13.200015],[0.000000,0.000000,1.000000,0.000000],[0,0,-1,0],[9E+09,9E+09,9E+09,9E+09,9E+09,9E+09]];
    CONST robtarget T1237:=[[80.000004,30.000000,13.200015],[0.000000,0.000000,1.000000,0.000000],[0,0,-1,0],[9E+09,9E+09,9E+09,9E+09,9E+09,9E+09]];
    CONST robtarget T1238:=[[81.260008,30.028279,13.200015],[0.000000,0.000000,1.000000,0.000000],[0,0,-1,0],[9E+09,9E+09,9E+09,9E+09,9E+09,9E+09]];
    CONST robtarget T1239:=[[81.260008,37.608991,13.200015],[0.000000,0.000000,1.000000,0.000000],[0,0,-1,0],[9E+09,9E+09,9E+09,9E+09,9E+09,9E+09]];
    CONST robtarget T1240:=[[81.260008,52.391011,13.200015],[0.000000,0.000000,1.000000,0.000000],[0,0,-1,0],[9E+09,9E+09,9E+09,9E+09,9E+09,9E+09]];
    CONST robtarget T1241:=[[81.260008,72.608994,13.200015],[0.000000,0.000000,1.000000,0.000000],[0,0,-1,0],[9E+09,9E+09,9E+09,9E+09,9E+09,9E+09]];
    CONST robtarget T1242:=[[81.260008,87.391014,13.200015],[0.000000,0.000000,1.000000,0.000000],[0,0,-1,0],[9E+09,9E+09,9E+09,9E+09,9E+09,9E+09]];
    CONST robtarget T1243:=[[81.260008,107.608996,13.200015],[0.000000,0.000000,1.000000,0.000000],[0,0,-1,0],[9E+09,9E+09,9E+09,9E+09,9E+09,9E+09]];
    CONST robtarget T1244:=[[81.260008,122.391017,13.200015],[0.000000,0.000000,1.000000,0.000000],[0,0,-1,0],[9E+09,9E+09,9E+09,9E+09,9E+09,9E+09]];
    CONST robtarget T1245:=[[81.260008,129.971729,13.200015],[0.000000,0.000000,1.000000,0.000000],[0,0,-1,0],[9E+09,9E+09,9E+09,9E+09,9E+09,9E+09]];
    CONST robtarget T1246:=[[82.520013,129.931001,13.200015],[0.000000,0.000000,1.000000,0.000000],[0,0,-1,0],[9E+09,9E+09,9E+09,9E+09,9E+09,9E+09]];
    CONST robtarget T1247:=[[82.520013,122.050628,13.200015],[0.000000,0.000000,1.000000,0.000000],[0,0,-1,0],[9E+09,9E+09,9E+09,9E+09,9E+09,9E+09]];
    CONST robtarget T1248:=[[82.520013,107.949384,13.200015],[0.000000,0.000000,1.000000,0.000000],[0,0,-1,0],[9E+09,9E+09,9E+09,9E+09,9E+09,9E+09]];
    CONST robtarget T1249:=[[82.520013,87.050626,13.200015],[0.000000,0.000000,1.000000,0.000000],[0,0,-1,0],[9E+09,9E+09,9E+09,9E+09,9E+09,9E+09]];
    CONST robtarget T1250:=[[82.520013,72.949381,13.200015],[0.000000,0.000000,1.000000,0.000000],[0,0,-1,0],[9E+09,9E+09,9E+09,9E+09,9E+09,9E+09]];
    CONST robtarget T1251:=[[82.520013,52.050624,13.200015],[0.000000,0.000000,1.000000,0.000000],[0,0,-1,0],[9E+09,9E+09,9E+09,9E+09,9E+09,9E+09]];
    CONST robtarget T1252:=[[82.520013,37.949379,13.200015],[0.000000,0.000000,1.000000,0.000000],[0,0,-1,0],[9E+09,9E+09,9E+09,9E+09,9E+09,9E+09]];
    CONST robtarget T1253:=[[82.520013,30.069007,13.200015],[0.000000,0.000000,1.000000,0.000000],[0,0,-1,0],[9E+09,9E+09,9E+09,9E+09,9E+09,9E+09]];
    CONST robtarget T1254:=[[83.780017,30.153959,13.200015],[0.000000,0.000000,1.000000,0.000000],[0,0,-1,0],[9E+09,9E+09,9E+09,9E+09,9E+09,9E+09]];
    CONST robtarget T1255:=[[83.780017,38.524551,13.200015],[0.000000,0.000000,1.000000,0.000000],[0,0,-1,0],[9E+09,9E+09,9E+09,9E+09,9E+09,9E+09]];
    CONST robtarget T1256:=[[83.780017,51.475451,13.200015],[0.000000,0.000000,1.000000,0.000000],[0,0,-1,0],[9E+09,9E+09,9E+09,9E+09,9E+09,9E+09]];
    CONST robtarget T1257:=[[83.780017,73.524553,13.200015],[0.000000,0.000000,1.000000,0.000000],[0,0,-1,0],[9E+09,9E+09,9E+09,9E+09,9E+09,9E+09]];
    CONST robtarget T1258:=[[83.780017,86.475455,13.200015],[0.000000,0.000000,1.000000,0.000000],[0,0,-1,0],[9E+09,9E+09,9E+09,9E+09,9E+09,9E+09]];
    CONST robtarget T1259:=[[83.780017,108.524556,13.200015],[0.000000,0.000000,1.000000,0.000000],[0,0,-1,0],[9E+09,9E+09,9E+09,9E+09,9E+09,9E+09]];
    CONST robtarget T1260:=[[83.780017,121.475457,13.200015],[0.000000,0.000000,1.000000,0.000000],[0,0,-1,0],[9E+09,9E+09,9E+09,9E+09,9E+09,9E+09]];
    CONST robtarget T1261:=[[83.780017,129.846049,13.200015],[0.000000,0.000000,1.000000,0.000000],[0,0,-1,0],[9E+09,9E+09,9E+09,9E+09,9E+09,9E+09]];
    CONST robtarget T1262:=[[85.040022,129.735844,13.200015],[0.000000,0.000000,1.000000,0.000000],[0,0,-1,0],[9E+09,9E+09,9E+09,9E+09,9E+09,9E+09]];
    CONST robtarget T1263:=[[85.040022,120.544921,13.200015],[0.000000,0.000000,1.000000,0.000000],[0,0,-1,0],[9E+09,9E+09,9E+09,9E+09,9E+09,9E+09]];
    CONST robtarget T1264:=[[85.040022,109.455091,13.200015],[0.000000,0.000000,1.000000,0.000000],[0,0,-1,0],[9E+09,9E+09,9E+09,9E+09,9E+09,9E+09]];
    CONST robtarget T1265:=[[85.040022,85.544918,13.200015],[0.000000,0.000000,1.000000,0.000000],[0,0,-1,0],[9E+09,9E+09,9E+09,9E+09,9E+09,9E+09]];
    CONST robtarget T1266:=[[85.040022,74.455090,13.200015],[0.000000,0.000000,1.000000,0.000000],[0,0,-1,0],[9E+09,9E+09,9E+09,9E+09,9E+09,9E+09]];
    CONST robtarget T1267:=[[85.040022,50.544916,13.200015],[0.000000,0.000000,1.000000,0.000000],[0,0,-1,0],[9E+09,9E+09,9E+09,9E+09,9E+09,9E+09]];
    CONST robtarget T1268:=[[85.040022,39.455086,13.200015],[0.000000,0.000000,1.000000,0.000000],[0,0,-1,0],[9E+09,9E+09,9E+09,9E+09,9E+09,9E+09]];
    CONST robtarget T1269:=[[85.040022,30.264163,13.200015],[0.000000,0.000000,1.000000,0.000000],[0,0,-1,0],[9E+09,9E+09,9E+09,9E+09,9E+09,9E+09]];
    CONST robtarget T1270:=[[86.300026,30.406130,13.200015],[0.000000,0.000000,1.000000,0.000000],[0,0,-1,0],[9E+09,9E+09,9E+09,9E+09,9E+09,9E+09]];
    CONST robtarget T1271:=[[86.300026,40.937335,13.200015],[0.000000,0.000000,1.000000,0.000000],[0,0,-1,0],[9E+09,9E+09,9E+09,9E+09,9E+09,9E+09]];
    CONST robtarget T1272:=[[86.300026,49.062665,13.200015],[0.000000,0.000000,1.000000,0.000000],[0,0,-1,0],[9E+09,9E+09,9E+09,9E+09,9E+09,9E+09]];
    CONST robtarget T1273:=[[86.300026,75.937339,13.200015],[0.000000,0.000000,1.000000,0.000000],[0,0,-1,0],[9E+09,9E+09,9E+09,9E+09,9E+09,9E+09]];
    CONST robtarget T1274:=[[86.300026,84.062668,13.200015],[0.000000,0.000000,1.000000,0.000000],[0,0,-1,0],[9E+09,9E+09,9E+09,9E+09,9E+09,9E+09]];
    CONST robtarget T1275:=[[86.300026,110.937342,13.200015],[0.000000,0.000000,1.000000,0.000000],[0,0,-1,0],[9E+09,9E+09,9E+09,9E+09,9E+09,9E+09]];
    CONST robtarget T1276:=[[86.300026,119.062672,13.200015],[0.000000,0.000000,1.000000,0.000000],[0,0,-1,0],[9E+09,9E+09,9E+09,9E+09,9E+09,9E+09]];
    CONST robtarget T1277:=[[86.300026,129.593877,13.200015],[0.000000,0.000000,1.000000,0.000000],[0,0,-1,0],[9E+09,9E+09,9E+09,9E+09,9E+09,9E+09]];
    CONST robtarget T1278:=[[87.560031,129.413129,13.200015],[0.000000,0.000000,1.000000,0.000000],[0,0,-1,0],[9E+09,9E+09,9E+09,9E+09,9E+09,9E+09]];
    CONST robtarget T1279:=[[87.560031,30.586879,13.200015],[0.000000,0.000000,1.000000,0.000000],[0,0,-1,0],[9E+09,9E+09,9E+09,9E+09,9E+09,9E+09]];
    CONST robtarget T1280:=[[88.820035,30.786444,13.200015],[0.000000,0.000000,1.000000,0.000000],[0,0,-1,0],[9E+09,9E+09,9E+09,9E+09,9E+09,9E+09]];
    CONST robtarget T1281:=[[88.820035,129.213563,13.200015],[0.000000,0.000000,1.000000,0.000000],[0,0,-1,0],[9E+09,9E+09,9E+09,9E+09,9E+09,9E+09]];
    CONST robtarget T1282:=[[90.080040,128.960575,13.200015],[0.000000,0.000000,1.000000,0.000000],[0,0,-1,0],[9E+09,9E+09,9E+09,9E+09,9E+09,9E+09]];
    CONST robtarget T1283:=[[90.080040,31.039433,13.200015],[0.000000,0.000000,1.000000,0.000000],[0,0,-1,0],[9E+09,9E+09,9E+09,9E+09,9E+09,9E+09]];
    CONST robtarget T1284:=[[91.340044,31.307526,13.200015],[0.000000,0.000000,1.000000,0.000000],[0,0,-1,0],[9E+09,9E+09,9E+09,9E+09,9E+09,9E+09]];
    CONST robtarget T1285:=[[91.340044,128.692481,13.200015],[0.000000,0.000000,1.000000,0.000000],[0,0,-1,0],[9E+09,9E+09,9E+09,9E+09,9E+09,9E+09]];
    CONST robtarget T1286:=[[92.600049,128.374988,13.200015],[0.000000,0.000000,1.000000,0.000000],[0,0,-1,0],[9E+09,9E+09,9E+09,9E+09,9E+09,9E+09]];
    CONST robtarget T1287:=[[92.600049,31.625019,13.200015],[0.000000,0.000000,1.000000,0.000000],[0,0,-1,0],[9E+09,9E+09,9E+09,9E+09,9E+09,9E+09]];
    CONST robtarget T1288:=[[93.860053,31.969479,13.200015],[0.000000,0.000000,1.000000,0.000000],[0,0,-1,0],[9E+09,9E+09,9E+09,9E+09,9E+09,9E+09]];
    CONST robtarget T1289:=[[93.860053,128.030529,13.200015],[0.000000,0.000000,1.000000,0.000000],[0,0,-1,0],[9E+09,9E+09,9E+09,9E+09,9E+09,9E+09]];
    CONST robtarget T1290:=[[95.120058,127.652167,13.200015],[0.000000,0.000000,1.000000,0.000000],[0,0,-1,0],[9E+09,9E+09,9E+09,9E+09,9E+09,9E+09]];
    CONST robtarget T1291:=[[95.120058,32.347841,13.200015],[0.000000,0.000000,1.000000,0.000000],[0,0,-1,0],[9E+09,9E+09,9E+09,9E+09,9E+09,9E+09]];
    CONST robtarget T1292:=[[96.380062,32.772318,13.200015],[0.000000,0.000000,1.000000,0.000000],[0,0,-1,0],[9E+09,9E+09,9E+09,9E+09,9E+09,9E+09]];
    CONST robtarget T1293:=[[96.380062,127.227690,13.200015],[0.000000,0.000000,1.000000,0.000000],[0,0,-1,0],[9E+09,9E+09,9E+09,9E+09,9E+09,9E+09]];
    CONST robtarget T1294:=[[97.640067,126.783143,13.200015],[0.000000,0.000000,1.000000,0.000000],[0,0,-1,0],[9E+09,9E+09,9E+09,9E+09,9E+09,9E+09]];
    CONST robtarget T1295:=[[97.640067,33.216864,13.200015],[0.000000,0.000000,1.000000,0.000000],[0,0,-1,0],[9E+09,9E+09,9E+09,9E+09,9E+09,9E+09]];
    CONST robtarget T1296:=[[98.900071,33.722290,13.200015],[0.000000,0.000000,1.000000,0.000000],[0,0,-1,0],[9E+09,9E+09,9E+09,9E+09,9E+09,9E+09]];
    CONST robtarget T1297:=[[98.900071,126.277717,13.200015],[0.000000,0.000000,1.000000,0.000000],[0,0,-1,0],[9E+09,9E+09,9E+09,9E+09,9E+09,9E+09]];
    CONST robtarget T1298:=[[100.160076,125.745278,13.200015],[0.000000,0.000000,1.000000,0.000000],[0,0,-1,0],[9E+09,9E+09,9E+09,9E+09,9E+09,9E+09]];
    CONST robtarget T1299:=[[100.160076,34.254730,13.200015],[0.000000,0.000000,1.000000,0.000000],[0,0,-1,0],[9E+09,9E+09,9E+09,9E+09,9E+09,9E+09]];
    CONST robtarget T1300:=[[101.420080,34.827050,13.200015],[0.000000,0.000000,1.000000,0.000000],[0,0,-1,0],[9E+09,9E+09,9E+09,9E+09,9E+09,9E+09]];
    CONST robtarget T1301:=[[101.420080,125.172958,13.200015],[0.000000,0.000000,1.000000,0.000000],[0,0,-1,0],[9E+09,9E+09,9E+09,9E+09,9E+09,9E+09]];
    CONST robtarget T1302:=[[102.680085,124.546114,13.200015],[0.000000,0.000000,1.000000,0.000000],[0,0,-1,0],[9E+09,9E+09,9E+09,9E+09,9E+09,9E+09]];
    CONST robtarget T1303:=[[102.680085,35.453894,13.200015],[0.000000,0.000000,1.000000,0.000000],[0,0,-1,0],[9E+09,9E+09,9E+09,9E+09,9E+09,9E+09]];
    CONST robtarget T1304:=[[103.940089,36.110177,13.200015],[0.000000,0.000000,1.000000,0.000000],[0,0,-1,0],[9E+09,9E+09,9E+09,9E+09,9E+09,9E+09]];
    CONST robtarget T1305:=[[103.940089,123.889831,13.200015],[0.000000,0.000000,1.000000,0.000000],[0,0,-1,0],[9E+09,9E+09,9E+09,9E+09,9E+09,9E+09]];
    CONST robtarget T1306:=[[105.200094,123.174878,13.200015],[0.000000,0.000000,1.000000,0.000000],[0,0,-1,0],[9E+09,9E+09,9E+09,9E+09,9E+09,9E+09]];
    CONST robtarget T1307:=[[105.200094,36.825129,13.200015],[0.000000,0.000000,1.000000,0.000000],[0,0,-1,0],[9E+09,9E+09,9E+09,9E+09,9E+09,9E+09]];
    CONST robtarget T1308:=[[106.460098,37.589739,13.200015],[0.000000,0.000000,1.000000,0.000000],[0,0,-1,0],[9E+09,9E+09,9E+09,9E+09,9E+09,9E+09]];
    CONST robtarget T1309:=[[106.460098,122.410268,13.200015],[0.000000,0.000000,1.000000,0.000000],[0,0,-1,0],[9E+09,9E+09,9E+09,9E+09,9E+09,9E+09]];
    CONST robtarget T1310:=[[107.720103,121.607260,13.200015],[0.000000,0.000000,1.000000,0.000000],[0,0,-1,0],[9E+09,9E+09,9E+09,9E+09,9E+09,9E+09]];
    CONST robtarget T1311:=[[107.720103,81.789524,13.200015],[0.000000,0.000000,1.000000,0.000000],[0,0,-1,0],[9E+09,9E+09,9E+09,9E+09,9E+09,9E+09]];
    CONST robtarget T1312:=[[107.720103,78.210483,13.200015],[0.000000,0.000000,1.000000,0.000000],[0,0,-1,0],[9E+09,9E+09,9E+09,9E+09,9E+09,9E+09]];
    CONST robtarget T1313:=[[107.720103,38.392748,13.200015],[0.000000,0.000000,1.000000,0.000000],[0,0,-1,0],[9E+09,9E+09,9E+09,9E+09,9E+09,9E+09]];
    CONST robtarget T1314:=[[108.980107,39.265681,13.200015],[0.000000,0.000000,1.000000,0.000000],[0,0,-1,0],[9E+09,9E+09,9E+09,9E+09,9E+09,9E+09]];
    CONST robtarget T1315:=[[108.980107,75.547902,13.200015],[0.000000,0.000000,1.000000,0.000000],[0,0,-1,0],[9E+09,9E+09,9E+09,9E+09,9E+09,9E+09]];
    CONST robtarget T1316:=[[108.980107,84.452106,13.200015],[0.000000,0.000000,1.000000,0.000000],[0,0,-1,0],[9E+09,9E+09,9E+09,9E+09,9E+09,9E+09]];
    CONST robtarget T1317:=[[108.980107,120.734326,13.200015],[0.000000,0.000000,1.000000,0.000000],[0,0,-1,0],[9E+09,9E+09,9E+09,9E+09,9E+09,9E+09]];
    CONST robtarget T1318:=[[110.240112,119.803025,13.200015],[0.000000,0.000000,1.000000,0.000000],[0,0,-1,0],[9E+09,9E+09,9E+09,9E+09,9E+09,9E+09]];
    CONST robtarget T1319:=[[110.240112,85.779969,13.200015],[0.000000,0.000000,1.000000,0.000000],[0,0,-1,0],[9E+09,9E+09,9E+09,9E+09,9E+09,9E+09]];
    CONST robtarget T1320:=[[110.240112,74.220038,13.200015],[0.000000,0.000000,1.000000,0.000000],[0,0,-1,0],[9E+09,9E+09,9E+09,9E+09,9E+09,9E+09]];
    CONST robtarget T1321:=[[110.240112,40.196983,13.200015],[0.000000,0.000000,1.000000,0.000000],[0,0,-1,0],[9E+09,9E+09,9E+09,9E+09,9E+09,9E+09]];
    CONST robtarget T1322:=[[111.500116,41.180273,13.200015],[0.000000,0.000000,1.000000,0.000000],[0,0,-1,0],[9E+09,9E+09,9E+09,9E+09,9E+09,9E+09]];
    CONST robtarget T1323:=[[111.500116,73.379202,13.200015],[0.000000,0.000000,1.000000,0.000000],[0,0,-1,0],[9E+09,9E+09,9E+09,9E+09,9E+09,9E+09]];
    CONST robtarget T1324:=[[111.500116,86.620805,13.200015],[0.000000,0.000000,1.000000,0.000000],[0,0,-1,0],[9E+09,9E+09,9E+09,9E+09,9E+09,9E+09]];
    CONST robtarget T1325:=[[111.500116,118.819735,13.200015],[0.000000,0.000000,1.000000,0.000000],[0,0,-1,0],[9E+09,9E+09,9E+09,9E+09,9E+09,9E+09]];
    CONST robtarget T1326:=[[112.760121,117.767805,13.200015],[0.000000,0.000000,1.000000,0.000000],[0,0,-1,0],[9E+09,9E+09,9E+09,9E+09,9E+09,9E+09]];
    CONST robtarget T1327:=[[112.760121,87.152583,13.200015],[0.000000,0.000000,1.000000,0.000000],[0,0,-1,0],[9E+09,9E+09,9E+09,9E+09,9E+09,9E+09]];
    CONST robtarget T1328:=[[112.760121,72.847425,13.200015],[0.000000,0.000000,1.000000,0.000000],[0,0,-1,0],[9E+09,9E+09,9E+09,9E+09,9E+09,9E+09]];
    CONST robtarget T1329:=[[112.760121,42.232203,13.200015],[0.000000,0.000000,1.000000,0.000000],[0,0,-1,0],[9E+09,9E+09,9E+09,9E+09,9E+09,9E+09]];
    CONST robtarget T1330:=[[114.020125,43.373063,13.200015],[0.000000,0.000000,1.000000,0.000000],[0,0,-1,0],[9E+09,9E+09,9E+09,9E+09,9E+09,9E+09]];
    CONST robtarget T1331:=[[114.020125,72.576253,13.200015],[0.000000,0.000000,1.000000,0.000000],[0,0,-1,0],[9E+09,9E+09,9E+09,9E+09,9E+09,9E+09]];
    CONST robtarget T1332:=[[114.020125,87.423755,13.200015],[0.000000,0.000000,1.000000,0.000000],[0,0,-1,0],[9E+09,9E+09,9E+09,9E+09,9E+09,9E+09]];
    CONST robtarget T1333:=[[114.020125,116.626944,13.200015],[0.000000,0.000000,1.000000,0.000000],[0,0,-1,0],[9E+09,9E+09,9E+09,9E+09,9E+09,9E+09]];
    CONST robtarget T1334:=[[115.280130,115.412758,13.200015],[0.000000,0.000000,1.000000,0.000000],[0,0,-1,0],[9E+09,9E+09,9E+09,9E+09,9E+09,9E+09]];
    CONST robtarget T1335:=[[115.280130,87.487316,13.200015],[0.000000,0.000000,1.000000,0.000000],[0,0,-1,0],[9E+09,9E+09,9E+09,9E+09,9E+09,9E+09]];
    CONST robtarget T1336:=[[115.280130,72.512692,13.200015],[0.000000,0.000000,1.000000,0.000000],[0,0,-1,0],[9E+09,9E+09,9E+09,9E+09,9E+09,9E+09]];
    CONST robtarget T1337:=[[115.280130,44.587250,13.200015],[0.000000,0.000000,1.000000,0.000000],[0,0,-1,0],[9E+09,9E+09,9E+09,9E+09,9E+09,9E+09]];
    CONST robtarget T1338:=[[116.540134,45.884908,13.200015],[0.000000,0.000000,1.000000,0.000000],[0,0,-1,0],[9E+09,9E+09,9E+09,9E+09,9E+09,9E+09]];
